LIN {X 0,Y 369.216,Z 142.49,A -85,B 0,C 180,E1 -12872.663,E2 -12872.663} C_VEL
LIN {X 0,Y 369.197,Z 142.498,A -85,B 0,C 180,E1 -12876.558,E2 -12876.558} C_VEL
LIN {X 0,Y 369.156,Z 142.497,A -85,B 0,C 180,E1 -12877.428,E2 -12877.428} C_VEL
LIN {X 0,Y 368.474,Z 142.588,A -85,B 0,C 180,E1 -12878.338,E2 -12878.338} C_VEL
LIN {X 0,Y 365.538,Z 142.949,A -85,B 0,C 180,E1 -12879.815,E2 -12879.815} C_VEL
LIN {X 0,Y 363.064,Z 143.259,A -85,B 0,C 180,E1 -12881.01,E2 -12881.01} C_VEL
LIN {X 0,Y 362.026,Z 143.387,A -85,B 0,C 180,E1 -12881.936,E2 -12881.936} C_VEL
LIN {X 0,Y 361.954,Z 143.398,A -85,B 0,C 180,E1 -12882.25,E2 -12882.25} C_VEL
LIN {X 0,Y 361.96,Z 143.399,A -85,B 0,C 180,E1 -12884.62,E2 -12884.62} C_VEL
LIN {X 0,Y 361.957,Z 143.398,A -85,B 0,C 180,E1 -12888.099,E2 -12888.099} C_VEL
LIN {X 0,Y 361.859,Z 143.407,A -85,B 0,C 180,E1 -12891.654,E2 -12891.654} C_VEL
LIN {X 0,Y 361.924,Z 143.399,A -85,B 0,C 180,E1 -12895.29,E2 -12895.29} C_VEL
LIN {X 0,Y 361.919,Z 143.401,A -85,B 0,C 180,E1 -12897.778,E2 -12897.778} C_VEL
LIN {X 0,Y 361.856,Z 143.409,A -85,B 0,C 180,E1 -12901.627,E2 -12901.627} C_VEL
LIN {X 0,Y 361.871,Z 143.406,A -85,B 0,C 180,E1 -12905.345,E2 -12905.345} C_VEL
LIN {X 0,Y 361.869,Z 143.406,A -85,B 0,C 180,E1 -12909.027,E2 -12909.027} C_VEL
LIN {X 0,Y 361.88,Z 143.406,A -85,B 0,C 180,E1 -12912.44,E2 -12912.44} C_VEL
LIN {X 0,Y 361.862,Z 143.411,A -85,B 0,C 180,E1 -12915.639,E2 -12915.639} C_VEL
LIN {X 0,Y 361.869,Z 143.407,A -85,B 0,C 180,E1 -12919.238,E2 -12919.238} C_VEL
LIN {X 0,Y 361.866,Z 143.407,A -85,B 0,C 180,E1 -12922.982,E2 -12922.982} C_VEL
LIN {X 0,Y 361.857,Z 143.407,A -85,B 0,C 180,E1 -12926.63,E2 -12926.63} C_VEL
LIN {X 0,Y 361.871,Z 143.41,A -85,B 0,C 180,E1 -12929.672,E2 -12929.672} C_VEL
LIN {X 0,Y 361.951,Z 143.401,A -85,B 0,C 180,E1 -12933.475,E2 -12933.475} C_VEL
LIN {X 0,Y 361.887,Z 143.407,A -85,B 0,C 180,E1 -12937.145,E2 -12937.145} C_VEL
LIN {X 0,Y 361.918,Z 143.401,A -85,B 0,C 180,E1 -12940.724,E2 -12940.724} C_VEL
LIN {X 0,Y 361.943,Z 143.396,A -85,B 0,C 180,E1 -12944.226,E2 -12944.226} C_VEL
LIN {X 0,Y 361.996,Z 143.391,A -85,B 0,C 180,E1 -12946.528,E2 -12946.528} C_VEL
LIN {X 0,Y 362.029,Z 143.386,A -85,B 0,C 180,E1 -12949.938,E2 -12949.938} C_VEL
LIN {X 0,Y 362.158,Z 143.373,A -85,B 0,C 180,E1 -12953.314,E2 -12953.314} C_VEL
LIN {X 0,Y 362.281,Z 143.354,A -85,B 0,C 180,E1 -12957.777,E2 -12957.777} C_VEL
LIN {X 0,Y 362.426,Z 143.336,A -85,B 0,C 180,E1 -12960,E2 -12960} C_VEL
LIN {X 0,Y 362.281,Z 143.355,A -85,B 0,C 180,E1 -12962.224,E2 -12962.224} C_VEL
LIN {X 0,Y 362.171,Z 143.374,A -85,B 0,C 180,E1 -12966.687,E2 -12966.687} C_VEL
LIN {X 0,Y 362.072,Z 143.384,A -85,B 0,C 180,E1 -12968.934,E2 -12968.934} C_VEL
LIN {X 0,Y 361.959,Z 143.398,A -85,B 0,C 180,E1 -12972.333,E2 -12972.333} C_VEL
LIN {X 0,Y 361.961,Z 143.4,A -85,B 0,C 180,E1 -12974.621,E2 -12974.621} C_VEL
LIN {X 0,Y 361.958,Z 143.397,A -85,B 0,C 180,E1 -12978.1,E2 -12978.1} C_VEL
LIN {X 0,Y 361.86,Z 143.407,A -85,B 0,C 180,E1 -12981.655,E2 -12981.655} C_VEL
LIN {X 0,Y 361.925,Z 143.398,A -85,B 0,C 180,E1 -12985.291,E2 -12985.291} C_VEL
LIN {X 0,Y 361.917,Z 143.401,A -85,B 0,C 180,E1 -12987.779,E2 -12987.779} C_VEL
LIN {X 0,Y 361.846,Z 143.408,A -85,B 0,C 180,E1 -12991.286,E2 -12991.286} C_VEL
LIN {X 0,Y 361.854,Z 143.412,A -85,B 0,C 180,E1 -12994.281,E2 -12994.281} C_VEL
LIN {X 0,Y 361.865,Z 143.406,A -85,B 0,C 180,E1 -12997.224,E2 -12997.224} C_VEL
LIN {X 0,Y 361.872,Z 143.405,A -85,B 0,C 180,E1 -13000.763,E2 -13000.763} C_VEL
LIN {X 0,Y 361.822,Z 143.413,A -85,B 0,C 180,E1 -13004.368,E2 -13004.368} C_VEL
LIN {X 0,Y 361.836,Z 143.413,A -85,B 0,C 180,E1 -13007.569,E2 -13007.569} C_VEL
LIN {X 0,Y 361.869,Z 143.406,A -85,B 0,C 180,E1 -13010.974,E2 -13010.974} C_VEL
LIN {X 0,Y 361.875,Z 143.405,A -85,B 0,C 180,E1 -13014.656,E2 -13014.656} C_VEL
LIN {X 0,Y 361.838,Z 143.412,A -85,B 0,C 180,E1 -13018.371,E2 -13018.371} C_VEL
LIN {X 0,Y 361.909,Z 143.415,A -85,B 0,C 180,E1 -13019.6,E2 -13019.6} C_VEL
LIN {X 0,Y 364.625,Z 156.408,A -85,B 0,C 180,E1 -13022.671,E2 -13022.671} C_VEL
LIN {X 0,Y 365.599,Z 162.364,A -85,B 0,C 180,E1 -13024.029,E2 -13024.029} C_VEL
LIN {X 0,Y 364.449,Z 176.387,A -85,B 0,C 180,E1 -13027.015,E2 -13027.015} C_VEL
LIN {X 0,Y 363.824,Z 184.769,A -85,B 0,C 180,E1 -13028.787,E2 -13028.787} C_VEL
LIN {X 0,Y 368.173,Z 221.285,A -85,B 0,C 180,E1 -13029.864,E2 -13029.864} C_VEL
LIN {X 0,Y 366.668,Z 294.38,A -85,B 0,C 180,E1 -13031.564,E2 -13031.564} C_VEL
LIN {X 0,Y 365.977,Z 308.139,A -85,B 0,C 180,E1 -13032.107,E2 -13032.107} C_VEL
LIN {X 0,Y 365.231,Z 320.13,A -85,B 0,C 180,E1 -13032.792,E2 -13032.792} C_VEL
LIN {X 0,Y 364.244,Z 332.659,A -85,B 0,C 180,E1 -13033.754,E2 -13033.754} C_VEL
LIN {X 0,Y 363.427,Z 343.96,A -85,B 0,C 180,E1 -13034.867,E2 -13034.867} C_VEL
LIN {X 0,Y 362.616,Z 353.865,A -85,B 0,C 180,E1 -13036.083,E2 -13036.083} C_VEL
LIN {X 0,Y 361.884,Z 364.213,A -85,B 0,C 180,E1 -13037.665,E2 -13037.665} C_VEL
LIN {X 0,Y 361.231,Z 371.672,A -85,B 0,C 180,E1 -13039.066,E2 -13039.066} C_VEL
LIN {X 0,Y 360.793,Z 378.999,A -85,B 0,C 180,E1 -13040.753,E2 -13040.753} C_VEL
LIN {X 0,Y 360.628,Z 383.937,A -85,B 0,C 180,E1 -13042.16,E2 -13042.16} C_VEL
LIN {X 0,Y 360.458,Z 388.862,A -85,B 0,C 180,E1 -13043.92,E2 -13043.92} C_VEL
LIN {X 0,Y 360.482,Z 392.245,A -85,B 0,C 180,E1 -13045.528,E2 -13045.528} C_VEL
LIN {X 0,Y 360.417,Z 393.997,A -85,B 0,C 180,E1 -13046.647,E2 -13046.647} C_VEL
LIN {X 0,Y 360.545,Z 395.32,A -85,B 0,C 180,E1 -13047.766,E2 -13047.766} C_VEL
LIN {X 0,Y 360.539,Z 396.212,A -85,B 0,C 180,E1 -13048.883,E2 -13048.883} C_VEL
LIN {X 0,Y 360.527,Z 396.662,A -85,B 0,C 180,E1 -13050,E2 -13050} C_VEL
LIN {X 0,Y 360.516,Z 396.658,A -85,B 0,C 180,E1 -13051.117,E2 -13051.117} C_VEL
LIN {X 0,Y 360.429,Z 396.239,A -85,B 0,C 180,E1 -13052.235,E2 -13052.235} C_VEL
LIN {X 0,Y 360.366,Z 395.415,A -85,B 0,C 180,E1 -13053.355,E2 -13053.355} C_VEL
LIN {X 0,Y 360.383,Z 394.141,A -85,B 0,C 180,E1 -13054.474,E2 -13054.474} C_VEL
LIN {X 0,Y 360.318,Z 391.949,A -85,B 0,C 180,E1 -13055.868,E2 -13055.868} C_VEL
LIN {X 0,Y 360.598,Z 387.648,A -85,B 0,C 180,E1 -13057.842,E2 -13057.842} C_VEL
LIN {X 0,Y 360.929,Z 382.737,A -85,B 0,C 180,E1 -13059.527,E2 -13059.527} C_VEL
LIN {X 0,Y 361.665,Z 375.38,A -85,B 0,C 180,E1 -13061.489,E2 -13061.489} C_VEL
LIN {X 0,Y 362.609,Z 367.453,A -85,B 0,C 180,E1 -13063.164,E2 -13063.164} C_VEL
LIN {X 0,Y 363.547,Z 358.621,A -85,B 0,C 180,E1 -13064.675,E2 -13064.675} C_VEL
LIN {X 0,Y 364.773,Z 348.543,A -85,B 0,C 180,E1 -13066.079,E2 -13066.079} C_VEL
LIN {X 0,Y 366.12,Z 337.576,A -85,B 0,C 180,E1 -13067.31,E2 -13067.31} C_VEL
LIN {X 0,Y 367.554,Z 325.219,A -85,B 0,C 180,E1 -13068.391,E2 -13068.391} C_VEL
LIN {X 0,Y 368.706,Z 312.247,A -85,B 0,C 180,E1 -13069.269,E2 -13069.269} C_VEL
LIN {X 0,Y 369.888,Z 298.194,A -85,B 0,C 180,E1 -13069.927,E2 -13069.927} C_VEL
LIN {X 0,Y 370.467,Z 285.445,A -85,B 0,C 180,E1 -13070.329,E2 -13070.329} C_VEL
LIN {X 0,Y 372.333,Z 220.719,A -85,B 0,C 180,E1 -13071.896,E2 -13071.896} C_VEL
LIN {X 0,Y 370.378,Z 204.902,A -85,B 0,C 180,E1 -13072.497,E2 -13072.497} C_VEL
LIN {X 0,Y 367.323,Z 188.483,A -85,B 0,C 180,E1 -13073.223,E2 -13073.223} C_VEL
LIN {X 0,Y 365.724,Z 180.687,A -85,B 0,C 180,E1 -13073.613,E2 -13073.613} C_VEL
LIN {X 0,Y 367.221,Z 166.298,A -85,B 0,C 180,E1 -13076.728,E2 -13076.728} C_VEL
LIN {X 0,Y 365.197,Z 156.175,A -85,B 0,C 180,E1 -13079.289,E2 -13079.289} C_VEL
LIN {X 0,Y 362.447,Z 145.496,A -85,B 0,C 180,E1 -13082.224,E2 -13082.224} C_VEL
LIN {X 0,Y 361.868,Z 143.412,A -85,B 0,C 180,E1 -13082.86,E2 -13082.86} C_VEL
LIN {X 0,Y 361.872,Z 143.409,A -85,B 0,C 180,E1 -13085.637,E2 -13085.637} C_VEL
LIN {X 0,Y 361.874,Z 143.41,A -85,B 0,C 180,E1 -13089.027,E2 -13089.027} C_VEL
LIN {X 0,Y 361.84,Z 143.413,A -85,B 0,C 180,E1 -13092.829,E2 -13092.829} C_VEL
LIN {X 0,Y 361.821,Z 143.412,A -85,B 0,C 180,E1 -13095.947,E2 -13095.947} C_VEL
LIN {X 0,Y 361.839,Z 143.408,A -85,B 0,C 180,E1 -13099.245,E2 -13099.245} C_VEL
LIN {X 0,Y 361.866,Z 143.404,A -85,B 0,C 180,E1 -13102.777,E2 -13102.777} C_VEL
LIN {X 0,Y 361.857,Z 143.404,A -85,B 0,C 180,E1 -13105.719,E2 -13105.719} C_VEL
LIN {X 0,Y 361.876,Z 143.408,A -85,B 0,C 180,E1 -13109.672,E2 -13109.672} C_VEL
LIN {X 0,Y 361.957,Z 143.396,A -85,B 0,C 180,E1 -13113.475,E2 -13113.475} C_VEL
LIN {X 0,Y 361.894,Z 143.402,A -85,B 0,C 180,E1 -13117.145,E2 -13117.145} C_VEL
LIN {X 0,Y 361.907,Z 143.404,A -85,B 0,C 180,E1 -13120.723,E2 -13120.723} C_VEL
LIN {X 0,Y 361.946,Z 143.396,A -85,B 0,C 180,E1 -13124.226,E2 -13124.226} C_VEL
LIN {X 0,Y 362.002,Z 143.391,A -85,B 0,C 180,E1 -13126.528,E2 -13126.528} C_VEL
LIN {X 0,Y 362.003,Z 143.393,A -85,B 0,C 180,E1 -13129.937,E2 -13129.937} C_VEL
LIN {X 0,Y 362.138,Z 143.38,A -85,B 0,C 180,E1 -13133.313,E2 -13133.313} C_VEL
LIN {X 0,Y 362.28,Z 143.363,A -85,B 0,C 180,E1 -13137.776,E2 -13137.776} C_VEL
LIN {X 0,Y 362.271,Z 143.399,A -85,B 0,C 180,E1 -13139.374,E2 -13139.374} C_VEL
LIN {X 0,Y 363.828,Z 149.687,A -85,B 0,C 180,E1 -13141.279,E2 -13141.279} C_VEL
LIN {X 0,Y 369.872,Z 162.966,A -85,B 0,C 180,E1 -13142.249,E2 -13142.249} C_VEL
LIN {X 0,Y 373.599,Z 171.886,A -85,B 0,C 180,E1 -13142.827,E2 -13142.827} C_VEL
LIN {X 0,Y 373.603,Z 177.913,A -85,B 0,C 180,E1 -13142.993,E2 -13142.993} C_VEL
LIN {X 0,Y 370.924,Z 256.422,A -85,B 0,C 180,E1 -13144.925,E2 -13144.925} C_VEL
LIN {X 0,Y 370.325,Z 269.377,A -85,B 0,C 180,E1 -13145.445,E2 -13145.445} C_VEL
LIN {X 0,Y 369.501,Z 282.588,A -85,B 0,C 180,E1 -13146.21,E2 -13146.21} C_VEL
LIN {X 0,Y 368.37,Z 295.305,A -85,B 0,C 180,E1 -13147.21,E2 -13147.21} C_VEL
LIN {X 0,Y 367.186,Z 306.94,A -85,B 0,C 180,E1 -13148.392,E2 -13148.392} C_VEL
LIN {X 0,Y 366.046,Z 316.914,A -85,B 0,C 180,E1 -13149.671,E2 -13149.671} C_VEL
LIN {X 0,Y 364.896,Z 326.008,A -85,B 0,C 180,E1 -13151.104,E2 -13151.104} C_VEL
LIN {X 0,Y 363.882,Z 333.5,A -85,B 0,C 180,E1 -13152.549,E2 -13152.549} C_VEL
LIN {X 0,Y 363.102,Z 339.353,A -85,B 0,C 180,E1 -13153.919,E2 -13153.919} C_VEL
LIN {X 0,Y 362.234,Z 345.726,A -85,B 0,C 180,E1 -13155.761,E2 -13155.761} C_VEL
LIN {X 0,Y 361.527,Z 350.802,A -85,B 0,C 180,E1 -13157.72,E2 -13157.72} C_VEL
LIN {X 0,Y 361.079,Z 353.856,A -85,B 0,C 180,E1 -13159.322,E2 -13159.322} C_VEL
LIN {X 0,Y 360.773,Z 355.83,A -85,B 0,C 180,E1 -13160.761,E2 -13160.761} C_VEL
LIN {X 0,Y 360.607,Z 356.736,A -85,B 0,C 180,E1 -13161.734,E2 -13161.734} C_VEL
LIN {X 0,Y 360.406,Z 357.591,A -85,B 0,C 180,E1 -13163.578,E2 -13163.578} C_VEL
LIN {X 0,Y 360.338,Z 357.323,A -85,B 0,C 180,E1 -13165.409,E2 -13165.409} C_VEL
LIN {X 0,Y 360.335,Z 356.51,A -85,B 0,C 180,E1 -13166.653,E2 -13166.653} C_VEL
LIN {X 0,Y 360.495,Z 354.072,A -85,B 0,C 180,E1 -13168.682,E2 -13168.682} C_VEL
LIN {X 0,Y 360.795,Z 350.782,A -85,B 0,C 180,E1 -13170.428,E2 -13170.428} C_VEL
LIN {X 0,Y 361.1,Z 345.75,A -85,B 0,C 180,E1 -13172.359,E2 -13172.359} C_VEL
LIN {X 0,Y 361.657,Z 339.068,A -85,B 0,C 180,E1 -13174.301,E2 -13174.301} C_VEL
LIN {X 0,Y 362.212,Z 331.861,A -85,B 0,C 180,E1 -13175.94,E2 -13175.94} C_VEL
LIN {X 0,Y 362.867,Z 323.153,A -85,B 0,C 180,E1 -13177.54,E2 -13177.54} C_VEL
LIN {X 0,Y 363.717,Z 313.001,A -85,B 0,C 180,E1 -13179.043,E2 -13179.043} C_VEL
LIN {X 0,Y 364.558,Z 301.376,A -85,B 0,C 180,E1 -13180.408,E2 -13180.408} C_VEL
LIN {X 0,Y 365.294,Z 291.019,A -85,B 0,C 180,E1 -13181.38,E2 -13181.38} C_VEL
LIN {X 0,Y 365.95,Z 279.585,A -85,B 0,C 180,E1 -13182.234,E2 -13182.234} C_VEL
LIN {X 0,Y 366.468,Z 266.205,A -85,B 0,C 180,E1 -13182.978,E2 -13182.978} C_VEL
LIN {X 0,Y 366.947,Z 253.458,A -85,B 0,C 180,E1 -13183.461,E2 -13183.461} C_VEL
LIN {X 0,Y 368.802,Z 168.805,A -85,B 0,C 180,E1 -13185.403,E2 -13185.403} C_VEL
LIN {X 0,Y 366.602,Z 159.202,A -85,B 0,C 180,E1 -13185.738,E2 -13185.738} C_VEL
LIN {X 0,Y 362.416,Z 146.013,A -85,B 0,C 180,E1 -13186.279,E2 -13186.279} C_VEL
LIN {X 0,Y 361.912,Z 143.405,A -85,B 0,C 180,E1 -13186.992,E2 -13186.992} C_VEL
LIN {X 0,Y 361.867,Z 143.406,A -85,B 0,C 180,E1 -13190.973,E2 -13190.973} C_VEL
LIN {X 0,Y 361.873,Z 143.405,A -85,B 0,C 180,E1 -13194.655,E2 -13194.655} C_VEL
LIN {X 0,Y 361.836,Z 143.41,A -85,B 0,C 180,E1 -13198.37,E2 -13198.37} C_VEL
LIN {X 0,Y 361.899,Z 143.403,A -85,B 0,C 180,E1 -13200.955,E2 -13200.955} C_VEL
LIN {X 0,Y 361.954,Z 143.4,A -85,B 0,C 180,E1 -13203.475,E2 -13203.475} C_VEL
LIN {X 0,Y 361.89,Z 143.408,A -85,B 0,C 180,E1 -13207.144,E2 -13207.144} C_VEL
LIN {X 0,Y 361.885,Z 143.405,A -85,B 0,C 180,E1 -13210.722,E2 -13210.722} C_VEL
LIN {X 0,Y 361.942,Z 143.396,A -85,B 0,C 180,E1 -13214.226,E2 -13214.226} C_VEL
LIN {X 0,Y 361.998,Z 143.391,A -85,B 0,C 180,E1 -13216.527,E2 -13216.527} C_VEL
LIN {X 0,Y 362.03,Z 143.385,A -85,B 0,C 180,E1 -13219.938,E2 -13219.938} C_VEL
LIN {X 0,Y 362.159,Z 143.372,A -85,B 0,C 180,E1 -13223.313,E2 -13223.313} C_VEL
LIN {X 0,Y 362.281,Z 143.354,A -85,B 0,C 180,E1 -13227.776,E2 -13227.776} C_VEL
LIN {X 0,Y 362.427,Z 143.336,A -85,B 0,C 180,E1 -13230,E2 -13230} C_VEL
LIN {X 0,Y 362.281,Z 143.356,A -85,B 0,C 180,E1 -13232.223,E2 -13232.223} C_VEL
LIN {X 0,Y 362.159,Z 143.376,A -85,B 0,C 180,E1 -13236.686,E2 -13236.686} C_VEL
LIN {X 0,Y 362.029,Z 143.387,A -85,B 0,C 180,E1 -13240.062,E2 -13240.062} C_VEL
LIN {X 0,Y 361.954,Z 143.398,A -85,B 0,C 180,E1 -13242.25,E2 -13242.25} C_VEL
LIN {X 0,Y 361.309,Z 143.484,A -85,B 0,C 180,E1 -13243.179,E2 -13243.179} C_VEL
LIN {X 0,Y 358.42,Z 143.841,A -85,B 0,C 180,E1 -13244.687,E2 -13244.687} C_VEL
LIN {X 0,Y 355.975,Z 144.141,A -85,B 0,C 180,E1 -13245.908,E2 -13245.908} C_VEL
LIN {X 0,Y 354.955,Z 144.269,A -85,B 0,C 180,E1 -13246.854,E2 -13246.854} C_VEL
LIN {X 0,Y 354.889,Z 144.275,A -85,B 0,C 180,E1 -13247.174,E2 -13247.174} C_VEL
LIN {X 0,Y 354.863,Z 144.279,A -85,B 0,C 180,E1 -13249.674,E2 -13249.674} C_VEL
LIN {X 0,Y 354.824,Z 144.283,A -85,B 0,C 180,E1 -13253.337,E2 -13253.337} C_VEL
LIN {X 0,Y 354.886,Z 144.276,A -85,B 0,C 180,E1 -13256.982,E2 -13256.982} C_VEL
LIN {X 0,Y 354.851,Z 144.281,A -85,B 0,C 180,E1 -13259.678,E2 -13259.678} C_VEL
LIN {X 0,Y 354.827,Z 144.285,A -85,B 0,C 180,E1 -13263.682,E2 -13263.682} C_VEL
LIN {X 0,Y 354.796,Z 144.289,A -85,B 0,C 180,E1 -13266.459,E2 -13266.459} C_VEL
LIN {X 0,Y 354.82,Z 144.285,A -85,B 0,C 180,E1 -13269.423,E2 -13269.423} C_VEL
LIN {X 0,Y 354.832,Z 144.282,A -85,B 0,C 180,E1 -13272.875,E2 -13272.875} C_VEL
LIN {X 0,Y 354.801,Z 144.289,A -85,B 0,C 180,E1 -13276.109,E2 -13276.109} C_VEL
LIN {X 0,Y 354.821,Z 144.285,A -85,B 0,C 180,E1 -13279.184,E2 -13279.184} C_VEL
LIN {X 0,Y 354.805,Z 144.286,A -85,B 0,C 180,E1 -13282.402,E2 -13282.402} C_VEL
LIN {X 0,Y 354.809,Z 144.286,A -85,B 0,C 180,E1 -13284.941,E2 -13284.941} C_VEL
LIN {X 0,Y 354.791,Z 144.287,A -85,B 0,C 180,E1 -13288.405,E2 -13288.405} C_VEL
LIN {X 0,Y 354.847,Z 144.285,A -85,B 0,C 180,E1 -13291.619,E2 -13291.619} C_VEL
LIN {X 0,Y 354.896,Z 144.275,A -85,B 0,C 180,E1 -13294.173,E2 -13294.173} C_VEL
LIN {X 0,Y 354.832,Z 144.284,A -85,B 0,C 180,E1 -13297.894,E2 -13297.894} C_VEL
LIN {X 0,Y 354.92,Z 144.272,A -85,B 0,C 180,E1 -13301.892,E2 -13301.892} C_VEL
LIN {X 0,Y 354.94,Z 144.269,A -85,B 0,C 180,E1 -13305.981,E2 -13305.981} C_VEL
LIN {X 0,Y 354.976,Z 144.265,A -85,B 0,C 180,E1 -13309.736,E2 -13309.736} C_VEL
LIN {X 0,Y 355.123,Z 144.25,A -85,B 0,C 180,E1 -13313.181,E2 -13313.181} C_VEL
LIN {X 0,Y 355.244,Z 144.231,A -85,B 0,C 180,E1 -13317.733,E2 -13317.733} C_VEL
LIN {X 0,Y 355.396,Z 144.212,A -85,B 0,C 180,E1 -13320,E2 -13320} C_VEL
LIN {X 0,Y 355.244,Z 144.232,A -85,B 0,C 180,E1 -13322.268,E2 -13322.268} C_VEL
LIN {X 0,Y 355.137,Z 144.249,A -85,B 0,C 180,E1 -13326.82,E2 -13326.82} C_VEL
LIN {X 0,Y 355.014,Z 144.262,A -85,B 0,C 180,E1 -13329.113,E2 -13329.113} C_VEL
LIN {X 0,Y 354.92,Z 144.277,A -85,B 0,C 180,E1 -13332.581,E2 -13332.581} C_VEL
LIN {X 0,Y 354.889,Z 144.277,A -85,B 0,C 180,E1 -13336.096,E2 -13336.096} C_VEL
LIN {X 0,Y 354.905,Z 144.279,A -85,B 0,C 180,E1 -13338.472,E2 -13338.472} C_VEL
LIN {X 0,Y 354.815,Z 144.288,A -85,B 0,C 180,E1 -13342.108,E2 -13342.108} C_VEL
LIN {X 0,Y 354.897,Z 144.276,A -85,B 0,C 180,E1 -13345.828,E2 -13345.828} C_VEL
LIN {X 0,Y 354.853,Z 144.281,A -85,B 0,C 180,E1 -13349.679,E2 -13349.679} C_VEL
LIN {X 0,Y 354.805,Z 144.287,A -85,B 0,C 180,E1 -13353.703,E2 -13353.703} C_VEL
LIN {X 0,Y 354.799,Z 144.289,A -85,B 0,C 180,E1 -13356.46,E2 -13356.46} C_VEL
LIN {X 0,Y 354.824,Z 144.284,A -85,B 0,C 180,E1 -13359.424,E2 -13359.424} C_VEL
LIN {X 0,Y 354.804,Z 144.286,A -85,B 0,C 180,E1 -13362.871,E2 -13362.871} C_VEL
LIN {X 0,Y 354.768,Z 144.294,A -85,B 0,C 180,E1 -13366.104,E2 -13366.104} C_VEL
LIN {X 0,Y 354.788,Z 144.288,A -85,B 0,C 180,E1 -13369.18,E2 -13369.18} C_VEL
LIN {X 0,Y 354.808,Z 144.286,A -85,B 0,C 180,E1 -13372.403,E2 -13372.403} C_VEL
LIN {X 0,Y 354.812,Z 144.285,A -85,B 0,C 180,E1 -13374.941,E2 -13374.941} C_VEL
LIN {X 0,Y 354.826,Z 144.287,A -85,B 0,C 180,E1 -13379.005,E2 -13379.005} C_VEL
LIN {X 0,Y 354.893,Z 144.446,A -85,B 0,C 180,E1 -13379.383,E2 -13379.383} C_VEL
LIN {X 0,Y 357.935,Z 159.065,A -85,B 0,C 180,E1 -13382.895,E2 -13382.895} C_VEL
LIN {X 0,Y 358.604,Z 164.655,A -85,B 0,C 180,E1 -13384.179,E2 -13384.179} C_VEL
LIN {X 0,Y 356.86,Z 184.383,A -85,B 0,C 180,E1 -13388.445,E2 -13388.445} C_VEL
LIN {X 0,Y 361.314,Z 221.994,A -85,B 0,C 180,E1 -13389.591,E2 -13389.591} C_VEL
LIN {X 0,Y 359.764,Z 294.104,A -85,B 0,C 180,E1 -13391.308,E2 -13391.308} C_VEL
LIN {X 0,Y 359.082,Z 307.818,A -85,B 0,C 180,E1 -13391.862,E2 -13391.862} C_VEL
LIN {X 0,Y 358.264,Z 320.276,A -85,B 0,C 180,E1 -13392.594,E2 -13392.594} C_VEL
LIN {X 0,Y 357.251,Z 332.695,A -85,B 0,C 180,E1 -13393.574,E2 -13393.574} C_VEL
LIN {X 0,Y 356.409,Z 343.919,A -85,B 0,C 180,E1 -13394.708,E2 -13394.708} C_VEL
LIN {X 0,Y 355.516,Z 354.668,A -85,B 0,C 180,E1 -13396.08,E2 -13396.08} C_VEL
LIN {X 0,Y 354.749,Z 364.889,A -85,B 0,C 180,E1 -13397.704,E2 -13397.704} C_VEL
LIN {X 0,Y 354.024,Z 373.445,A -85,B 0,C 180,E1 -13399.419,E2 -13399.419} C_VEL
LIN {X 0,Y 353.682,Z 380.33,A -85,B 0,C 180,E1 -13401.142,E2 -13401.142} C_VEL
LIN {X 0,Y 353.397,Z 386.57,A -85,B 0,C 180,E1 -13403.147,E2 -13403.147} C_VEL
LIN {X 0,Y 353.384,Z 390.579,A -85,B 0,C 180,E1 -13404.866,E2 -13404.866} C_VEL
LIN {X 0,Y 353.335,Z 393.476,A -85,B 0,C 180,E1 -13406.579,E2 -13406.579} C_VEL
LIN {X 0,Y 353.447,Z 394.825,A -85,B 0,C 180,E1 -13407.721,E2 -13407.721} C_VEL
LIN {X 0,Y 353.475,Z 395.745,A -85,B 0,C 180,E1 -13408.861,E2 -13408.861} C_VEL
LIN {X 0,Y 353.462,Z 396.241,A -85,B 0,C 180,E1 -13410,E2 -13410} C_VEL
LIN {X 0,Y 353.432,Z 396.269,A -85,B 0,C 180,E1 -13411.14,E2 -13411.14} C_VEL
LIN {X 0,Y 353.33,Z 395.877,A -85,B 0,C 180,E1 -13412.28,E2 -13412.28} C_VEL
LIN {X 0,Y 353.282,Z 395.078,A -85,B 0,C 180,E1 -13413.422,E2 -13413.422} C_VEL
LIN {X 0,Y 353.289,Z 393.855,A -85,B 0,C 180,E1 -13414.564,E2 -13414.564} C_VEL
LIN {X 0,Y 353.235,Z 391.94,A -85,B 0,C 180,E1 -13415.838,E2 -13415.838} C_VEL
LIN {X 0,Y 353.53,Z 387.454,A -85,B 0,C 180,E1 -13417.999,E2 -13417.999} C_VEL
LIN {X 0,Y 353.908,Z 382.601,A -85,B 0,C 180,E1 -13419.718,E2 -13419.718} C_VEL
LIN {X 0,Y 354.688,Z 375.317,A -85,B 0,C 180,E1 -13421.719,E2 -13421.719} C_VEL
LIN {X 0,Y 355.689,Z 367.504,A -85,B 0,C 180,E1 -13423.425,E2 -13423.425} C_VEL
LIN {X 0,Y 356.694,Z 358.553,A -85,B 0,C 180,E1 -13425.009,E2 -13425.009} C_VEL
LIN {X 0,Y 358.122,Z 347.778,A -85,B 0,C 180,E1 -13426.533,E2 -13426.533} C_VEL
LIN {X 0,Y 359.558,Z 336.707,A -85,B 0,C 180,E1 -13427.783,E2 -13427.783} C_VEL
LIN {X 0,Y 361.039,Z 324.241,A -85,B 0,C 180,E1 -13428.883,E2 -13428.883} C_VEL
LIN {X 0,Y 362.179,Z 312.245,A -85,B 0,C 180,E1 -13429.704,E2 -13429.704} C_VEL
LIN {X 0,Y 363.414,Z 298.533,A -85,B 0,C 180,E1 -13430.371,E2 -13430.371} C_VEL
LIN {X 0,Y 364.071,Z 285.149,A -85,B 0,C 180,E1 -13430.813,E2 -13430.813} C_VEL
LIN {X 0,Y 366.037,Z 221.315,A -85,B 0,C 180,E1 -13432.406,E2 -13432.406} C_VEL
LIN {X 0,Y 364.169,Z 206.128,A -85,B 0,C 180,E1 -13433,E2 -13433} C_VEL
LIN {X 0,Y 360.866,Z 188.359,A -85,B 0,C 180,E1 -13433.827,E2 -13433.827} C_VEL
LIN {X 0,Y 359.191,Z 180.15,A -85,B 0,C 180,E1 -13434.261,E2 -13434.261} C_VEL
LIN {X 0,Y 360.437,Z 167.993,A -85,B 0,C 180,E1 -13436.959,E2 -13436.959} C_VEL
LIN {X 0,Y 358.62,Z 158.852,A -85,B 0,C 180,E1 -13439.337,E2 -13439.337} C_VEL
LIN {X 0,Y 356.06,Z 148.667,A -85,B 0,C 180,E1 -13442.204,E2 -13442.204} C_VEL
LIN {X 0,Y 354.815,Z 144.29,A -85,B 0,C 180,E1 -13443.558,E2 -13443.558} C_VEL
LIN {X 0,Y 354.802,Z 144.291,A -85,B 0,C 180,E1 -13446.459,E2 -13446.459} C_VEL
LIN {X 0,Y 354.828,Z 144.289,A -85,B 0,C 180,E1 -13449.424,E2 -13449.424} C_VEL
LIN {X 0,Y 354.792,Z 144.291,A -85,B 0,C 180,E1 -13452.867,E2 -13452.867} C_VEL
LIN {X 0,Y 354.77,Z 144.29,A -85,B 0,C 180,E1 -13456.104,E2 -13456.104} C_VEL
LIN {X 0,Y 354.791,Z 144.285,A -85,B 0,C 180,E1 -13459.179,E2 -13459.179} C_VEL
LIN {X 0,Y 354.81,Z 144.284,A -85,B 0,C 180,E1 -13462.403,E2 -13462.403} C_VEL
LIN {X 0,Y 354.815,Z 144.284,A -85,B 0,C 180,E1 -13464.941,E2 -13464.941} C_VEL
LIN {X 0,Y 354.796,Z 144.283,A -85,B 0,C 180,E1 -13468.405,E2 -13468.405} C_VEL
LIN {X 0,Y 354.85,Z 144.279,A -85,B 0,C 180,E1 -13471.618,E2 -13471.618} C_VEL
LIN {X 0,Y 354.903,Z 144.27,A -85,B 0,C 180,E1 -13474.172,E2 -13474.172} C_VEL
LIN {X 0,Y 354.838,Z 144.284,A -85,B 0,C 180,E1 -13477.894,E2 -13477.894} C_VEL
LIN {X 0,Y 354.893,Z 144.272,A -85,B 0,C 180,E1 -13481.908,E2 -13481.908} C_VEL
LIN {X 0,Y 354.946,Z 144.271,A -85,B 0,C 180,E1 -13485.981,E2 -13485.981} C_VEL
LIN {X 0,Y 354.959,Z 144.271,A -85,B 0,C 180,E1 -13489.735,E2 -13489.735} C_VEL
LIN {X 0,Y 355.103,Z 144.257,A -85,B 0,C 180,E1 -13493.18,E2 -13493.18} C_VEL
LIN {X 0,Y 355.243,Z 144.239,A -85,B 0,C 180,E1 -13497.732,E2 -13497.732} C_VEL
LIN {X 0,Y 355.213,Z 144.411,A -85,B 0,C 180,E1 -13498.724,E2 -13498.724} C_VEL
LIN {X 0,Y 356.811,Z 150.318,A -85,B 0,C 180,E1 -13500.585,E2 -13500.585} C_VEL
LIN {X 0,Y 362.801,Z 162.829,A -85,B 0,C 180,E1 -13501.572,E2 -13501.572} C_VEL
LIN {X 0,Y 367.561,Z 173.93,A -85,B 0,C 180,E1 -13502.353,E2 -13502.353} C_VEL
LIN {X 0,Y 364.521,Z 257.464,A -85,B 0,C 180,E1 -13504.457,E2 -13504.457} C_VEL
LIN {X 0,Y 363.854,Z 270.838,A -85,B 0,C 180,E1 -13505.021,E2 -13505.021} C_VEL
LIN {X 0,Y 363.039,Z 283.148,A -85,B 0,C 180,E1 -13505.763,E2 -13505.763} C_VEL
LIN {X 0,Y 361.943,Z 294.792,A -85,B 0,C 180,E1 -13506.69,E2 -13506.69} C_VEL
LIN {X 0,Y 360.745,Z 306.127,A -85,B 0,C 180,E1 -13507.838,E2 -13507.838} C_VEL
LIN {X 0,Y 359.513,Z 316.389,A -85,B 0,C 180,E1 -13509.139,E2 -13509.139} C_VEL
LIN {X 0,Y 358.295,Z 325.525,A -85,B 0,C 180,E1 -13510.575,E2 -13510.575} C_VEL
LIN {X 0,Y 357.088,Z 333.981,A -85,B 0,C 180,E1 -13512.214,E2 -13512.214} C_VEL
LIN {X 0,Y 356.184,Z 340.164,A -85,B 0,C 180,E1 -13513.696,E2 -13513.696} C_VEL
LIN {X 0,Y 355.302,Z 346.173,A -85,B 0,C 180,E1 -13515.487,E2 -13515.487} C_VEL
LIN {X 0,Y 354.612,Z 350.816,A -85,B 0,C 180,E1 -13517.294,E2 -13517.294} C_VEL
LIN {X 0,Y 354.231,Z 353.249,A -85,B 0,C 180,E1 -13518.508,E2 -13518.508} C_VEL
LIN {X 0,Y 353.896,Z 355.204,A -85,B 0,C 180,E1 -13519.73,E2 -13519.73} C_VEL
LIN {X 0,Y 353.669,Z 356.604,A -85,B 0,C 180,E1 -13520.958,E2 -13520.958} C_VEL
LIN {X 0,Y 353.455,Z 357.558,A -85,B 0,C 180,E1 -13522.196,E2 -13522.196} C_VEL
LIN {X 0,Y 353.325,Z 358.027,A -85,B 0,C 180,E1 -13523.795,E2 -13523.795} C_VEL
LIN {X 0,Y 353.265,Z 357.401,A -85,B 0,C 180,E1 -13525.955,E2 -13525.955} C_VEL
LIN {X 0,Y 353.262,Z 356.292,A -85,B 0,C 180,E1 -13527.23,E2 -13527.23} C_VEL
LIN {X 0,Y 353.476,Z 353.932,A -85,B 0,C 180,E1 -13528.974,E2 -13528.974} C_VEL
LIN {X 0,Y 353.798,Z 349.651,A -85,B 0,C 180,E1 -13531.096,E2 -13531.096} C_VEL
LIN {X 0,Y 354.165,Z 344.306,A -85,B 0,C 180,E1 -13532.998,E2 -13532.998} C_VEL
LIN {X 0,Y 354.678,Z 338.05,A -85,B 0,C 180,E1 -13534.728,E2 -13534.728} C_VEL
LIN {X 0,Y 355.31,Z 330.531,A -85,B 0,C 180,E1 -13536.398,E2 -13536.398} C_VEL
LIN {X 0,Y 356.062,Z 321.295,A -85,B 0,C 180,E1 -13538.047,E2 -13538.047} C_VEL
LIN {X 0,Y 356.899,Z 311.06,A -85,B 0,C 180,E1 -13539.513,E2 -13539.513} C_VEL
LIN {X 0,Y 357.736,Z 300.029,A -85,B 0,C 180,E1 -13540.784,E2 -13540.784} C_VEL
LIN {X 0,Y 358.465,Z 288.447,A -85,B 0,C 180,E1 -13541.839,E2 -13541.839} C_VEL
LIN {X 0,Y 359.192,Z 276.338,A -85,B 0,C 180,E1 -13542.694,E2 -13542.694} C_VEL
LIN {X 0,Y 359.723,Z 263.241,A -85,B 0,C 180,E1 -13543.373,E2 -13543.373} C_VEL
LIN {X 0,Y 360.143,Z 249.733,A -85,B 0,C 180,E1 -13543.829,E2 -13543.829} C_VEL
LIN {X 0,Y 361.987,Z 169.715,A -85,B 0,C 180,E1 -13545.701,E2 -13545.701} C_VEL
LIN {X 0,Y 359.87,Z 160.803,A -85,B 0,C 180,E1 -13546.023,E2 -13546.023} C_VEL
LIN {X 0,Y 355.276,Z 146.363,A -85,B 0,C 180,E1 -13546.629,E2 -13546.629} C_VEL
LIN {X 0,Y 354.855,Z 144.285,A -85,B 0,C 180,E1 -13547.212,E2 -13547.212} C_VEL
LIN {X 0,Y 354.815,Z 144.284,A -85,B 0,C 180,E1 -13550.666,E2 -13550.666} C_VEL
LIN {X 0,Y 354.821,Z 144.284,A -85,B 0,C 180,E1 -13554.3,E2 -13554.3} C_VEL
LIN {X 0,Y 354.786,Z 144.292,A -85,B 0,C 180,E1 -13557.666,E2 -13557.666} C_VEL
LIN {X 0,Y 354.868,Z 144.278,A -85,B 0,C 180,E1 -13560.621,E2 -13560.621} C_VEL
LIN {X 0,Y 354.899,Z 144.274,A -85,B 0,C 180,E1 -13564.172,E2 -13564.172} C_VEL
LIN {X 0,Y 354.834,Z 144.283,A -85,B 0,C 180,E1 -13567.894,E2 -13567.894} C_VEL
LIN {X 0,Y 354.888,Z 144.276,A -85,B 0,C 180,E1 -13571.907,E2 -13571.907} C_VEL
LIN {X 0,Y 354.941,Z 144.269,A -85,B 0,C 180,E1 -13575.981,E2 -13575.981} C_VEL
LIN {X 0,Y 354.977,Z 144.265,A -85,B 0,C 180,E1 -13579.735,E2 -13579.735} C_VEL
LIN {X 0,Y 355.124,Z 144.25,A -85,B 0,C 180,E1 -13583.18,E2 -13583.18} C_VEL
LIN {X 0,Y 355.244,Z 144.231,A -85,B 0,C 180,E1 -13587.732,E2 -13587.732} C_VEL
LIN {X 0,Y 355.396,Z 144.212,A -85,B 0,C 180,E1 -13590,E2 -13590} C_VEL
LIN {X 0,Y 355.244,Z 144.232,A -85,B 0,C 180,E1 -13592.267,E2 -13592.267} C_VEL
LIN {X 0,Y 355.123,Z 144.25,A -85,B 0,C 180,E1 -13596.819,E2 -13596.819} C_VEL
LIN {X 0,Y 354.976,Z 144.267,A -85,B 0,C 180,E1 -13600.264,E2 -13600.264} C_VEL
LIN {X 0,Y 354.94,Z 144.27,A -85,B 0,C 180,E1 -13604.019,E2 -13604.019} C_VEL
LIN {X 0,Y 354.889,Z 144.275,A -85,B 0,C 180,E1 -13607.174,E2 -13607.174} C_VEL
LIN {X 0,Y 354.255,Z 144.359,A -85,B 0,C 180,E1 -13608.121,E2 -13608.121} C_VEL
LIN {X 0,Y 351.364,Z 144.716,A -85,B 0,C 180,E1 -13609.66,E2 -13609.66} C_VEL
LIN {X 0,Y 348.891,Z 145.024,A -85,B 0,C 180,E1 -13610.905,E2 -13610.905} C_VEL
LIN {X 0,Y 347.833,Z 145.156,A -85,B 0,C 180,E1 -13611.87,E2 -13611.87} C_VEL
LIN {X 0,Y 347.751,Z 145.165,A -85,B 0,C 180,E1 -13612.197,E2 -13612.197} C_VEL
LIN {X 0,Y 347.808,Z 145.157,A -85,B 0,C 180,E1 -13615.108,E2 -13615.108} C_VEL
LIN {X 0,Y 347.809,Z 145.158,A -85,B 0,C 180,E1 -13617.693,E2 -13617.693} C_VEL
LIN {X 0,Y 347.767,Z 145.166,A -85,B 0,C 180,E1 -13620.346,E2 -13620.346} C_VEL
LIN {X 0,Y 347.745,Z 145.171,A -85,B 0,C 180,E1 -13624.044,E2 -13624.044} C_VEL
LIN {X 0,Y 347.759,Z 145.164,A -85,B 0,C 180,E1 -13627.32,E2 -13627.32} C_VEL
LIN {X 0,Y 347.79,Z 145.162,A -85,B 0,C 180,E1 -13630.288,E2 -13630.288} C_VEL
LIN {X 0,Y 347.783,Z 145.162,A -85,B 0,C 180,E1 -13633.398,E2 -13633.398} C_VEL
LIN {X 0,Y 347.766,Z 145.163,A -85,B 0,C 180,E1 -13636.679,E2 -13636.679} C_VEL
LIN {X 0,Y 347.754,Z 145.166,A -85,B 0,C 180,E1 -13640.171,E2 -13640.171} C_VEL
LIN {X 0,Y 347.768,Z 145.165,A -85,B 0,C 180,E1 -13643.935,E2 -13643.935} C_VEL
LIN {X 0,Y 347.739,Z 145.166,A -85,B 0,C 180,E1 -13646.929,E2 -13646.929} C_VEL
LIN {X 0,Y 347.801,Z 145.159,A -85,B 0,C 180,E1 -13650.99,E2 -13650.99} C_VEL
LIN {X 0,Y 347.829,Z 145.159,A -85,B 0,C 180,E1 -13653.608,E2 -13653.608} C_VEL
LIN {X 0,Y 347.785,Z 145.16,A -85,B 0,C 180,E1 -13656.162,E2 -13656.162} C_VEL
LIN {X 0,Y 347.814,Z 145.157,A -85,B 0,C 180,E1 -13659.91,E2 -13659.91} C_VEL
LIN {X 0,Y 347.864,Z 145.15,A -85,B 0,C 180,E1 -13662.36,E2 -13662.36} C_VEL
LIN {X 0,Y 347.894,Z 145.147,A -85,B 0,C 180,E1 -13665.971,E2 -13665.971} C_VEL
LIN {X 0,Y 347.926,Z 145.145,A -85,B 0,C 180,E1 -13669.526,E2 -13669.526} C_VEL
LIN {X 0,Y 348.089,Z 145.128,A -85,B 0,C 180,E1 -13673.042,E2 -13673.042} C_VEL
LIN {X 0,Y 348.206,Z 145.108,A -85,B 0,C 180,E1 -13677.687,E2 -13677.687} C_VEL
LIN {X 0,Y 348.344,Z 145.09,A -85,B 0,C 180,E1 -13680,E2 -13680} C_VEL
LIN {X 0,Y 348.206,Z 145.109,A -85,B 0,C 180,E1 -13682.314,E2 -13682.314} C_VEL
LIN {X 0,Y 348.105,Z 145.124,A -85,B 0,C 180,E1 -13686.958,E2 -13686.958} C_VEL
LIN {X 0,Y 347.966,Z 145.138,A -85,B 0,C 180,E1 -13689.299,E2 -13689.299} C_VEL
LIN {X 0,Y 347.889,Z 145.151,A -85,B 0,C 180,E1 -13692.84,E2 -13692.84} C_VEL
LIN {X 0,Y 347.838,Z 145.159,A -85,B 0,C 180,E1 -13696.432,E2 -13696.432} C_VEL
LIN {X 0,Y 347.854,Z 145.154,A -85,B 0,C 180,E1 -13698.861,E2 -13698.861} C_VEL
LIN {X 0,Y 347.761,Z 145.167,A -85,B 0,C 180,E1 -13702.581,E2 -13702.581} C_VEL
LIN {X 0,Y 347.81,Z 145.157,A -85,B 0,C 180,E1 -13705.109,E2 -13705.109} C_VEL
LIN {X 0,Y 347.81,Z 145.158,A -85,B 0,C 180,E1 -13707.694,E2 -13707.694} C_VEL
LIN {X 0,Y 347.763,Z 145.168,A -85,B 0,C 180,E1 -13710.347,E2 -13710.347} C_VEL
LIN {X 0,Y 347.744,Z 145.168,A -85,B 0,C 180,E1 -13714.464,E2 -13714.464} C_VEL
LIN {X 0,Y 347.776,Z 145.167,A -85,B 0,C 180,E1 -13717.99,E2 -13717.99} C_VEL
LIN {X 0,Y 347.766,Z 145.167,A -85,B 0,C 180,E1 -13721.828,E2 -13721.828} C_VEL
LIN {X 0,Y 347.708,Z 145.17,A -85,B 0,C 180,E1 -13725.027,E2 -13725.027} C_VEL
LIN {X 0,Y 347.75,Z 145.166,A -85,B 0,C 180,E1 -13728.398,E2 -13728.398} C_VEL
LIN {X 0,Y 347.774,Z 145.165,A -85,B 0,C 180,E1 -13732.012,E2 -13732.012} C_VEL
LIN {X 0,Y 347.745,Z 145.17,A -85,B 0,C 180,E1 -13735.537,E2 -13735.537} C_VEL
LIN {X 0,Y 347.835,Z 145.305,A -85,B 0,C 180,E1 -13739.114,E2 -13739.114} C_VEL
LIN {X 0,Y 350.756,Z 159.323,A -85,B 0,C 180,E1 -13742.559,E2 -13742.559} C_VEL
LIN {X 0,Y 351.645,Z 165.066,A -85,B 0,C 180,E1 -13743.916,E2 -13743.916} C_VEL
LIN {X 0,Y 350.099,Z 181.664,A -85,B 0,C 180,E1 -13747.579,E2 -13747.579} C_VEL
LIN {X 0,Y 349.911,Z 184.076,A -85,B 0,C 180,E1 -13748.11,E2 -13748.11} C_VEL
LIN {X 0,Y 354.458,Z 222.465,A -85,B 0,C 180,E1 -13749.305,E2 -13749.305} C_VEL
LIN {X 0,Y 352.875,Z 293.485,A -85,B 0,C 180,E1 -13751.042,E2 -13751.042} C_VEL
LIN {X 0,Y 352.176,Z 307.235,A -85,B 0,C 180,E1 -13751.606,E2 -13751.606} C_VEL
LIN {X 0,Y 351.39,Z 319.248,A -85,B 0,C 180,E1 -13752.317,E2 -13752.317} C_VEL
LIN {X 0,Y 350.426,Z 331.004,A -85,B 0,C 180,E1 -13753.244,E2 -13753.244} C_VEL
LIN {X 0,Y 349.46,Z 342.445,A -85,B 0,C 180,E1 -13754.397,E2 -13754.397} C_VEL
LIN {X 0,Y 348.535,Z 353.218,A -85,B 0,C 180,E1 -13755.76,E2 -13755.76} C_VEL
LIN {X 0,Y 347.817,Z 362.143,A -85,B 0,C 180,E1 -13757.158,E2 -13757.158} C_VEL
LIN {X 0,Y 347.205,Z 369.837,A -85,B 0,C 180,E1 -13758.618,E2 -13758.618} C_VEL
LIN {X 0,Y 346.716,Z 377.376,A -85,B 0,C 180,E1 -13760.374,E2 -13760.374} C_VEL
LIN {X 0,Y 346.493,Z 382.462,A -85,B 0,C 180,E1 -13761.838,E2 -13761.838} C_VEL
LIN {X 0,Y 346.298,Z 387.357,A -85,B 0,C 180,E1 -13763.592,E2 -13763.592} C_VEL
LIN {X 0,Y 346.341,Z 391.065,A -85,B 0,C 180,E1 -13765.345,E2 -13765.345} C_VEL
LIN {X 0,Y 346.255,Z 392.936,A -85,B 0,C 180,E1 -13766.509,E2 -13766.509} C_VEL
LIN {X 0,Y 346.35,Z 394.318,A -85,B 0,C 180,E1 -13767.675,E2 -13767.675} C_VEL
LIN {X 0,Y 346.412,Z 395.272,A -85,B 0,C 180,E1 -13768.838,E2 -13768.838} C_VEL
LIN {X 0,Y 346.398,Z 395.803,A -85,B 0,C 180,E1 -13770,E2 -13770} C_VEL
LIN {X 0,Y 346.35,Z 395.882,A -85,B 0,C 180,E1 -13771.163,E2 -13771.163} C_VEL
LIN {X 0,Y 346.233,Z 395.515,A -85,B 0,C 180,E1 -13772.327,E2 -13772.327} C_VEL
LIN {X 0,Y 346.201,Z 394.742,A -85,B 0,C 180,E1 -13773.492,E2 -13773.492} C_VEL
LIN {X 0,Y 346.198,Z 393.557,A -85,B 0,C 180,E1 -13774.658,E2 -13774.658} C_VEL
LIN {X 0,Y 346.212,Z 390.919,A -85,B 0,C 180,E1 -13776.411,E2 -13776.411} C_VEL
LIN {X 0,Y 346.481,Z 387.259,A -85,B 0,C 180,E1 -13778.163,E2 -13778.163} C_VEL
LIN {X 0,Y 346.875,Z 382.491,A -85,B 0,C 180,E1 -13779.917,E2 -13779.917} C_VEL
LIN {X 0,Y 347.524,Z 376.48,A -85,B 0,C 180,E1 -13781.668,E2 -13781.668} C_VEL
LIN {X 0,Y 348.572,Z 368.986,A -85,B 0,C 180,E1 -13783.407,E2 -13783.407} C_VEL
LIN {X 0,Y 349.697,Z 359.736,A -85,B 0,C 180,E1 -13785.146,E2 -13785.146} C_VEL
LIN {X 0,Y 351.028,Z 350.277,A -85,B 0,C 180,E1 -13786.577,E2 -13786.577} C_VEL
LIN {X 0,Y 352.664,Z 338.57,A -85,B 0,C 180,E1 -13787.993,E2 -13787.993} C_VEL
LIN {X 0,Y 354.216,Z 326.897,A -85,B 0,C 180,E1 -13789.11,E2 -13789.11} C_VEL
LIN {X 0,Y 355.438,Z 314.72,A -85,B 0,C 180,E1 -13790.018,E2 -13790.018} C_VEL
LIN {X 0,Y 356.823,Z 300.886,A -85,B 0,C 180,E1 -13790.765,E2 -13790.765} C_VEL
LIN {X 0,Y 357.615,Z 287.747,A -85,B 0,C 180,E1 -13791.244,E2 -13791.244} C_VEL
LIN {X 0,Y 359.821,Z 222.511,A -85,B 0,C 180,E1 -13792.913,E2 -13792.913} C_VEL
LIN {X 0,Y 357.994,Z 207.298,A -85,B 0,C 180,E1 -13793.537,E2 -13793.537} C_VEL
LIN {X 0,Y 354.992,Z 190.713,A -85,B 0,C 180,E1 -13794.332,E2 -13794.332} C_VEL
LIN {X 0,Y 352.598,Z 179.646,A -85,B 0,C 180,E1 -13794.941,E2 -13794.941} C_VEL
LIN {X 0,Y 353.627,Z 171.672,A -85,B 0,C 180,E1 -13796.741,E2 -13796.741} C_VEL
LIN {X 0,Y 353.448,Z 168.451,A -85,B 0,C 180,E1 -13797.536,E2 -13797.536} C_VEL
LIN {X 0,Y 351.571,Z 159.399,A -85,B 0,C 180,E1 -13799.984,E2 -13799.984} C_VEL
LIN {X 0,Y 349.483,Z 151.226,A -85,B 0,C 180,E1 -13802.369,E2 -13802.369} C_VEL
LIN {X 0,Y 347.769,Z 145.166,A -85,B 0,C 180,E1 -13804.331,E2 -13804.331} C_VEL
LIN {X 0,Y 347.778,Z 145.167,A -85,B 0,C 180,E1 -13807.989,E2 -13807.989} C_VEL
LIN {X 0,Y 347.754,Z 145.167,A -85,B 0,C 180,E1 -13811.83,E2 -13811.83} C_VEL
LIN {X 0,Y 347.709,Z 145.173,A -85,B 0,C 180,E1 -13815.027,E2 -13815.027} C_VEL
LIN {X 0,Y 347.754,Z 145.161,A -85,B 0,C 180,E1 -13818.397,E2 -13818.397} C_VEL
LIN {X 0,Y 347.776,Z 145.162,A -85,B 0,C 180,E1 -13822.011,E2 -13822.011} C_VEL
LIN {X 0,Y 347.748,Z 145.162,A -85,B 0,C 180,E1 -13825.536,E2 -13825.536} C_VEL
LIN {X 0,Y 347.748,Z 145.161,A -85,B 0,C 180,E1 -13828.3,E2 -13828.3} C_VEL
LIN {X 0,Y 347.782,Z 145.161,A -85,B 0,C 180,E1 -13830.987,E2 -13830.987} C_VEL
LIN {X 0,Y 347.834,Z 145.153,A -85,B 0,C 180,E1 -13833.608,E2 -13833.608} C_VEL
LIN {X 0,Y 347.792,Z 145.161,A -85,B 0,C 180,E1 -13836.162,E2 -13836.162} C_VEL
LIN {X 0,Y 347.815,Z 145.155,A -85,B 0,C 180,E1 -13839.909,E2 -13839.909} C_VEL
LIN {X 0,Y 347.835,Z 145.156,A -85,B 0,C 180,E1 -13843.568,E2 -13843.568} C_VEL
LIN {X 0,Y 347.893,Z 145.149,A -85,B 0,C 180,E1 -13847.16,E2 -13847.16} C_VEL
LIN {X 0,Y 347.938,Z 145.144,A -85,B 0,C 180,E1 -13850.7,E2 -13850.7} C_VEL
LIN {X 0,Y 348.071,Z 145.132,A -85,B 0,C 180,E1 -13853.041,E2 -13853.041} C_VEL
LIN {X 0,Y 348.196,Z 145.288,A -85,B 0,C 180,E1 -13857.975,E2 -13857.975} C_VEL
LIN {X 0,Y 349.85,Z 150.992,A -85,B 0,C 180,E1 -13859.838,E2 -13859.838} C_VEL
LIN {X 0,Y 356.439,Z 164.419,A -85,B 0,C 180,E1 -13860.984,E2 -13860.984} C_VEL
LIN {X 0,Y 361.322,Z 175.793,A -85,B 0,C 180,E1 -13861.818,E2 -13861.818} C_VEL
LIN {X 0,Y 358.176,Z 258.476,A -85,B 0,C 180,E1 -13863.973,E2 -13863.973} C_VEL
LIN {X 0,Y 357.45,Z 272.337,A -85,B 0,C 180,E1 -13864.581,E2 -13864.581} C_VEL
LIN {X 0,Y 356.506,Z 284.853,A -85,B 0,C 180,E1 -13865.373,E2 -13865.373} C_VEL
LIN {X 0,Y 355.307,Z 297.02,A -85,B 0,C 180,E1 -13866.388,E2 -13866.388} C_VEL
LIN {X 0,Y 354.057,Z 307.818,A -85,B 0,C 180,E1 -13867.536,E2 -13867.536} C_VEL
LIN {X 0,Y 352.725,Z 317.921,A -85,B 0,C 180,E1 -13868.883,E2 -13868.883} C_VEL
LIN {X 0,Y 351.429,Z 326.976,A -85,B 0,C 180,E1 -13870.368,E2 -13870.368} C_VEL
LIN {X 0,Y 350.311,Z 334.461,A -85,B 0,C 180,E1 -13871.866,E2 -13871.866} C_VEL
LIN {X 0,Y 349.161,Z 341.745,A -85,B 0,C 180,E1 -13873.68,E2 -13873.68} C_VEL
LIN {X 0,Y 348.388,Z 346.649,A -85,B 0,C 180,E1 -13875.203,E2 -13875.203} C_VEL
LIN {X 0,Y 347.632,Z 351.287,A -85,B 0,C 180,E1 -13877.046,E2 -13877.046} C_VEL
LIN {X 0,Y 347.036,Z 354.727,A -85,B 0,C 180,E1 -13878.906,E2 -13878.906} C_VEL
LIN {X 0,Y 346.553,Z 357.336,A -85,B 0,C 180,E1 -13881.113,E2 -13881.113} C_VEL
LIN {X 0,Y 346.304,Z 358.245,A -85,B 0,C 180,E1 -13882.68,E2 -13882.68} C_VEL
LIN {X 0,Y 346.234,Z 358.457,A -85,B 0,C 180,E1 -13884.016,E2 -13884.016} C_VEL
LIN {X 0,Y 346.169,Z 358.129,A -85,B 0,C 180,E1 -13885.235,E2 -13885.235} C_VEL
LIN {X 0,Y 346.17,Z 357.161,A -85,B 0,C 180,E1 -13886.709,E2 -13886.709} C_VEL
LIN {X 0,Y 346.217,Z 355.946,A -85,B 0,C 180,E1 -13887.832,E2 -13887.832} C_VEL
LIN {X 0,Y 346.521,Z 352.807,A -85,B 0,C 180,E1 -13889.811,E2 -13889.811} C_VEL
LIN {X 0,Y 346.839,Z 348.318,A -85,B 0,C 180,E1 -13891.792,E2 -13891.792} C_VEL
LIN {X 0,Y 347.233,Z 343.086,A -85,B 0,C 180,E1 -13893.543,E2 -13893.543} C_VEL
LIN {X 0,Y 347.717,Z 336.999,A -85,B 0,C 180,E1 -13895.172,E2 -13895.172} C_VEL
LIN {X 0,Y 348.445,Z 328.982,A -85,B 0,C 180,E1 -13896.895,E2 -13896.895} C_VEL
LIN {X 0,Y 349.265,Z 319.156,A -85,B 0,C 180,E1 -13898.593,E2 -13898.593} C_VEL
LIN {X 0,Y 350.102,Z 309.256,A -85,B 0,C 180,E1 -13899.968,E2 -13899.968} C_VEL
LIN {X 0,Y 350.907,Z 298.242,A -85,B 0,C 180,E1 -13901.201,E2 -13901.201} C_VEL
LIN {X 0,Y 351.695,Z 286.449,A -85,B 0,C 180,E1 -13902.25,E2 -13902.25} C_VEL
LIN {X 0,Y 352.428,Z 274.232,A -85,B 0,C 180,E1 -13903.078,E2 -13903.078} C_VEL
LIN {X 0,Y 352.863,Z 261.789,A -85,B 0,C 180,E1 -13903.699,E2 -13903.699} C_VEL
LIN {X 0,Y 353.275,Z 248.606,A -85,B 0,C 180,E1 -13904.129,E2 -13904.129} C_VEL
LIN {X 0,Y 355.185,Z 170.729,A -85,B 0,C 180,E1 -13905.991,E2 -13905.991} C_VEL
LIN {X 0,Y 353.158,Z 162.489,A -85,B 0,C 180,E1 -13906.297,E2 -13906.297} C_VEL
LIN {X 0,Y 348.106,Z 146.733,A -85,B 0,C 180,E1 -13906.973,E2 -13906.973} C_VEL
LIN {X 0,Y 347.797,Z 145.164,A -85,B 0,C 180,E1 -13907.444,E2 -13907.444} C_VEL
LIN {X 0,Y 347.751,Z 145.166,A -85,B 0,C 180,E1 -13911.207,E2 -13911.207} C_VEL
LIN {X 0,Y 347.788,Z 145.161,A -85,B 0,C 180,E1 -13914.124,E2 -13914.124} C_VEL
LIN {X 0,Y 347.737,Z 145.167,A -85,B 0,C 180,E1 -13918.086,E2 -13918.086} C_VEL
LIN {X 0,Y 347.804,Z 145.16,A -85,B 0,C 180,E1 -13920.99,E2 -13920.99} C_VEL
LIN {X 0,Y 347.831,Z 145.158,A -85,B 0,C 180,E1 -13923.607,E2 -13923.607} C_VEL
LIN {X 0,Y 347.788,Z 145.16,A -85,B 0,C 180,E1 -13926.161,E2 -13926.161} C_VEL
LIN {X 0,Y 347.804,Z 145.158,A -85,B 0,C 180,E1 -13929.908,E2 -13929.908} C_VEL
LIN {X 0,Y 347.831,Z 145.157,A -85,B 0,C 180,E1 -13933.568,E2 -13933.568} C_VEL
LIN {X 0,Y 347.889,Z 145.153,A -85,B 0,C 180,E1 -13937.16,E2 -13937.16} C_VEL
LIN {X 0,Y 347.963,Z 145.141,A -85,B 0,C 180,E1 -13940.701,E2 -13940.701} C_VEL
LIN {X 0,Y 348.09,Z 145.127,A -85,B 0,C 180,E1 -13943.042,E2 -13943.042} C_VEL
LIN {X 0,Y 348.207,Z 145.108,A -85,B 0,C 180,E1 -13947.686,E2 -13947.686} C_VEL
LIN {X 0,Y 348.345,Z 145.09,A -85,B 0,C 180,E1 -13950,E2 -13950} C_VEL
LIN {X 0,Y 348.206,Z 145.109,A -85,B 0,C 180,E1 -13952.313,E2 -13952.313} C_VEL
LIN {X 0,Y 348.09,Z 145.125,A -85,B 0,C 180,E1 -13956.958,E2 -13956.958} C_VEL
LIN {X 0,Y 347.927,Z 145.147,A -85,B 0,C 180,E1 -13960.474,E2 -13960.474} C_VEL
LIN {X 0,Y 347.896,Z 145.149,A -85,B 0,C 180,E1 -13964.149,E2 -13964.149} C_VEL
LIN {X 0,Y 347.889,Z 145.152,A -85,B 0,C 180,E1 -13968.29,E2 -13968.29} C_VEL
LIN {X 0,Y 347.751,Z 145.165,A -85,B 0,C 180,E1 -13972.197,E2 -13972.197} C_VEL
LIN {X 0,Y 347.106,Z 145.248,A -85,B 0,C 180,E1 -13973.164,E2 -13973.164} C_VEL
LIN {X 0,Y 344.304,Z 145.597,A -85,B 0,C 180,E1 -13974.739,E2 -13974.739} C_VEL
LIN {X 0,Y 341.913,Z 145.895,A -85,B 0,C 180,E1 -13976.013,E2 -13976.013} C_VEL
LIN {X 0,Y 340.874,Z 146.022,A -85,B 0,C 180,E1 -13976.999,E2 -13976.999} C_VEL
LIN {X 0,Y 340.782,Z 146.032,A -85,B 0,C 180,E1 -13977.332,E2 -13977.332} C_VEL
LIN {X 0,Y 340.762,Z 146.039,A -85,B 0,C 180,E1 -13979.978,E2 -13979.978} C_VEL
LIN {X 0,Y 340.692,Z 146.047,A -85,B 0,C 180,E1 -13983.846,E2 -13983.846} C_VEL
LIN {X 0,Y 340.702,Z 146.043,A -85,B 0,C 180,E1 -13986.741,E2 -13986.741} C_VEL
LIN {X 0,Y 340.76,Z 146.038,A -85,B 0,C 180,E1 -13990.262,E2 -13990.262} C_VEL
LIN {X 0,Y 340.732,Z 146.044,A -85,B 0,C 180,E1 -13993.788,E2 -13993.788} C_VEL
LIN {X 0,Y 340.73,Z 146.043,A -85,B 0,C 180,E1 -13997.948,E2 -13997.948} C_VEL
LIN {X 0,Y 340.735,Z 146.044,A -85,B 0,C 180,E1 -14001.774,E2 -14001.774} C_VEL
LIN {X 0,Y 340.719,Z 146.046,A -85,B 0,C 180,E1 -14005.595,E2 -14005.595} C_VEL
LIN {X 0,Y 340.701,Z 146.044,A -85,B 0,C 180,E1 -14008.956,E2 -14008.956} C_VEL
LIN {X 0,Y 340.775,Z 146.033,A -85,B 0,C 180,E1 -14012.474,E2 -14012.474} C_VEL
LIN {X 0,Y 340.753,Z 146.04,A -85,B 0,C 180,E1 -14015.639,E2 -14015.639} C_VEL
LIN {X 0,Y 340.746,Z 146.041,A -85,B 0,C 180,E1 -14019.475,E2 -14019.475} C_VEL
LIN {X 0,Y 340.855,Z 146.024,A -85,B 0,C 180,E1 -14021.985,E2 -14021.985} C_VEL
LIN {X 0,Y 340.866,Z 146.023,A -85,B 0,C 180,E1 -14025.705,E2 -14025.705} C_VEL
LIN {X 0,Y 340.868,Z 146.026,A -85,B 0,C 180,E1 -14029.307,E2 -14029.307} C_VEL
LIN {X 0,Y 341.057,Z 146.003,A -85,B 0,C 180,E1 -14032.898,E2 -14032.898} C_VEL
LIN {X 0,Y 341.168,Z 145.985,A -85,B 0,C 180,E1 -14037.639,E2 -14037.639} C_VEL
LIN {X 0,Y 341.295,Z 145.969,A -85,B 0,C 180,E1 -14040,E2 -14040} C_VEL
LIN {X 0,Y 341.168,Z 145.986,A -85,B 0,C 180,E1 -14042.362,E2 -14042.362} C_VEL
LIN {X 0,Y 341.074,Z 145.998,A -85,B 0,C 180,E1 -14047.102,E2 -14047.102} C_VEL
LIN {X 0,Y 340.869,Z 146.027,A -85,B 0,C 180,E1 -14050.694,E2 -14050.694} C_VEL
LIN {X 0,Y 340.861,Z 146.026,A -85,B 0,C 180,E1 -14054.325,E2 -14054.325} C_VEL
LIN {X 0,Y 340.837,Z 146.032,A -85,B 0,C 180,E1 -14058.467,E2 -14058.467} C_VEL
LIN {X 0,Y 340.716,Z 146.042,A -85,B 0,C 180,E1 -14061.842,E2 -14061.842} C_VEL
LIN {X 0,Y 340.771,Z 146.035,A -85,B 0,C 180,E1 -14065.665,E2 -14065.665} C_VEL
LIN {X 0,Y 340.74,Z 146.043,A -85,B 0,C 180,E1 -14068.32,E2 -14068.32} C_VEL
LIN {X 0,Y 340.703,Z 146.042,A -85,B 0,C 180,E1 -14071.045,E2 -14071.045} C_VEL
LIN {X 0,Y 340.718,Z 146.041,A -85,B 0,C 180,E1 -14075.279,E2 -14075.279} C_VEL
LIN {X 0,Y 340.717,Z 146.043,A -85,B 0,C 180,E1 -14078.388,E2 -14078.388} C_VEL
LIN {X 0,Y 340.731,Z 146.044,A -85,B 0,C 180,E1 -14082.052,E2 -14082.052} C_VEL
LIN {X 0,Y 340.652,Z 146.051,A -85,B 0,C 180,E1 -14086.227,E2 -14086.227} C_VEL
LIN {X 0,Y 340.689,Z 146.05,A -85,B 0,C 180,E1 -14089.754,E2 -14089.754} C_VEL
LIN {X 0,Y 340.705,Z 146.044,A -85,B 0,C 180,E1 -14093.259,E2 -14093.259} C_VEL
LIN {X 0,Y 340.693,Z 146.045,A -85,B 0,C 180,E1 -14096.154,E2 -14096.154} C_VEL
LIN {X 0,Y 340.738,Z 146.103,A -85,B 0,C 180,E1 -14098.831,E2 -14098.831} C_VEL
LIN {X 0,Y 343.639,Z 159.814,A -85,B 0,C 180,E1 -14102.272,E2 -14102.272} C_VEL
LIN {X 0,Y 344.655,Z 166.111,A -85,B 0,C 180,E1 -14103.796,E2 -14103.796} C_VEL
LIN {X 0,Y 342.965,Z 183.666,A -85,B 0,C 180,E1 -14107.748,E2 -14107.748} C_VEL
LIN {X 0,Y 347.606,Z 223.549,A -85,B 0,C 180,E1 -14109.035,E2 -14109.035} C_VEL
LIN {X 0,Y 345.969,Z 292.776,A -85,B 0,C 180,E1 -14110.764,E2 -14110.764} C_VEL
LIN {X 0,Y 345.274,Z 306.609,A -85,B 0,C 180,E1 -14111.34,E2 -14111.34} C_VEL
LIN {X 0,Y 344.431,Z 319.196,A -85,B 0,C 180,E1 -14112.101,E2 -14112.101} C_VEL
LIN {X 0,Y 343.444,Z 330.878,A -85,B 0,C 180,E1 -14113.047,E2 -14113.047} C_VEL
LIN {X 0,Y 342.455,Z 342.275,A -85,B 0,C 180,E1 -14114.222,E2 -14114.222} C_VEL
LIN {X 0,Y 341.512,Z 352.567,A -85,B 0,C 180,E1 -14115.547,E2 -14115.547} C_VEL
LIN {X 0,Y 340.823,Z 361.066,A -85,B 0,C 180,E1 -14116.89,E2 -14116.89} C_VEL
LIN {X 0,Y 340.211,Z 368.883,A -85,B 0,C 180,E1 -14118.381,E2 -14118.381} C_VEL
LIN {X 0,Y 339.656,Z 376.521,A -85,B 0,C 180,E1 -14120.172,E2 -14120.172} C_VEL
LIN {X 0,Y 339.429,Z 381.699,A -85,B 0,C 180,E1 -14121.667,E2 -14121.667} C_VEL
LIN {X 0,Y 339.228,Z 386.677,A -85,B 0,C 180,E1 -14123.458,E2 -14123.458} C_VEL
LIN {X 0,Y 339.248,Z 390.459,A -85,B 0,C 180,E1 -14125.247,E2 -14125.247} C_VEL
LIN {X 0,Y 339.179,Z 392.378,A -85,B 0,C 180,E1 -14126.437,E2 -14126.437} C_VEL
LIN {X 0,Y 339.254,Z 393.812,A -85,B 0,C 180,E1 -14127.626,E2 -14127.626} C_VEL
LIN {X 0,Y 339.35,Z 394.799,A -85,B 0,C 180,E1 -14128.814,E2 -14128.814} C_VEL
LIN {X 0,Y 339.336,Z 395.36,A -85,B 0,C 180,E1 -14130,E2 -14130} C_VEL
LIN {X 0,Y 339.255,Z 395.49,A -85,B 0,C 180,E1 -14131.187,E2 -14131.187} C_VEL
LIN {X 0,Y 339.137,Z 395.152,A -85,B 0,C 180,E1 -14132.376,E2 -14132.376} C_VEL
LIN {X 0,Y 339.121,Z 394.409,A -85,B 0,C 180,E1 -14133.565,E2 -14133.565} C_VEL
LIN {X 0,Y 339.076,Z 391.904,A -85,B 0,C 180,E1 -14135.789,E2 -14135.789} C_VEL
LIN {X 0,Y 339.325,Z 388.424,A -85,B 0,C 180,E1 -14137.737,E2 -14137.737} C_VEL
LIN {X 0,Y 339.687,Z 384.099,A -85,B 0,C 180,E1 -14139.528,E2 -14139.528} C_VEL
LIN {X 0,Y 340.404,Z 377.517,A -85,B 0,C 180,E1 -14141.613,E2 -14141.613} C_VEL
LIN {X 0,Y 341.461,Z 370.399,A -85,B 0,C 180,E1 -14143.389,E2 -14143.389} C_VEL
LIN {X 0,Y 342.511,Z 362.298,A -85,B 0,C 180,E1 -14145.042,E2 -14145.042} C_VEL
LIN {X 0,Y 343.948,Z 352.673,A -85,B 0,C 180,E1 -14146.623,E2 -14146.623} C_VEL
LIN {X 0,Y 345.522,Z 341.753,A -85,B 0,C 180,E1 -14148.071,E2 -14148.071} C_VEL
LIN {X 0,Y 347.142,Z 330.926,A -85,B 0,C 180,E1 -14149.208,E2 -14149.208} C_VEL
LIN {X 0,Y 348.521,Z 319.023,A -85,B 0,C 180,E1 -14150.202,E2 -14150.202} C_VEL
LIN {X 0,Y 349.991,Z 305.676,A -85,B 0,C 180,E1 -14151.035,E2 -14151.035} C_VEL
LIN {X 0,Y 351.022,Z 292.115,A -85,B 0,C 180,E1 -14151.625,E2 -14151.625} C_VEL
LIN {X 0,Y 352.257,Z 262.776,A -85,B 0,C 180,E1 -14152.42,E2 -14152.42} C_VEL
LIN {X 0,Y 353.629,Z 222.955,A -85,B 0,C 180,E1 -14153.48,E2 -14153.48} C_VEL
LIN {X 0,Y 351.657,Z 206.968,A -85,B 0,C 180,E1 -14154.168,E2 -14154.168} C_VEL
LIN {X 0,Y 348.498,Z 190.066,A -85,B 0,C 180,E1 -14155.03,E2 -14155.03} C_VEL
LIN {X 0,Y 346.101,Z 179.051,A -85,B 0,C 180,E1 -14155.685,E2 -14155.685} C_VEL
LIN {X 0,Y 346.956,Z 172.411,A -85,B 0,C 180,E1 -14157.226,E2 -14157.226} C_VEL
LIN {X 0,Y 345.413,Z 163.836,A -85,B 0,C 180,E1 -14159.565,E2 -14159.565} C_VEL
LIN {X 0,Y 343.289,Z 155.052,A -85,B 0,C 180,E1 -14162.16,E2 -14162.16} C_VEL
LIN {X 0,Y 340.717,Z 146.045,A -85,B 0,C 180,E1 -14165.156,E2 -14165.156} C_VEL
LIN {X 0,Y 340.713,Z 146.045,A -85,B 0,C 180,E1 -14168.386,E2 -14168.386} C_VEL
LIN {X 0,Y 340.703,Z 146.044,A -85,B 0,C 180,E1 -14172.045,E2 -14172.045} C_VEL
LIN {X 0,Y 340.655,Z 146.048,A -85,B 0,C 180,E1 -14176.227,E2 -14176.227} C_VEL
LIN {X 0,Y 340.692,Z 146.046,A -85,B 0,C 180,E1 -14179.753,E2 -14179.753} C_VEL
LIN {X 0,Y 340.708,Z 146.037,A -85,B 0,C 180,E1 -14183.258,E2 -14183.258} C_VEL
LIN {X 0,Y 340.696,Z 146.038,A -85,B 0,C 180,E1 -14186.153,E2 -14186.153} C_VEL
LIN {X 0,Y 340.745,Z 146.039,A -85,B 0,C 180,E1 -14190.329,E2 -14190.329} C_VEL
LIN {X 0,Y 340.807,Z 146.035,A -85,B 0,C 180,E1 -14193.02,E2 -14193.02} C_VEL
LIN {X 0,Y 340.76,Z 146.039,A -85,B 0,C 180,E1 -14195.638,E2 -14195.638} C_VEL
LIN {X 0,Y 340.755,Z 146.034,A -85,B 0,C 180,E1 -14199.474,E2 -14199.474} C_VEL
LIN {X 0,Y 340.796,Z 146.028,A -85,B 0,C 180,E1 -14201.98,E2 -14201.98} C_VEL
LIN {X 0,Y 340.873,Z 146.025,A -85,B 0,C 180,E1 -14205.705,E2 -14205.705} C_VEL
LIN {X 0,Y 340.851,Z 146.027,A -85,B 0,C 180,E1 -14209.305,E2 -14209.305} C_VEL
LIN {X 0,Y 341.019,Z 146.009,A -85,B 0,C 180,E1 -14212.897,E2 -14212.897} C_VEL
LIN {X 0,Y 341.041,Z 146.125,A -85,B 0,C 180,E1 -14217.12,E2 -14217.12} C_VEL
LIN {X 0,Y 342.688,Z 151.569,A -85,B 0,C 180,E1 -14219.008,E2 -14219.008} C_VEL
LIN {X 0,Y 346.816,Z 159.285,A -85,B 0,C 180,E1 -14219.763,E2 -14219.763} C_VEL
LIN {X 0,Y 351.734,Z 169.608,A -85,B 0,C 180,E1 -14220.653,E2 -14220.653} C_VEL
LIN {X 0,Y 355.254,Z 178.015,A -85,B 0,C 180,E1 -14221.283,E2 -14221.283} C_VEL
LIN {X 0,Y 351.927,Z 258.727,A -85,B 0,C 180,E1 -14223.434,E2 -14223.434} C_VEL
LIN {X 0,Y 351.186,Z 271.851,A -85,B 0,C 180,E1 -14224.016,E2 -14224.016} C_VEL
LIN {X 0,Y 350.286,Z 283.592,A -85,B 0,C 180,E1 -14224.747,E2 -14224.747} C_VEL
LIN {X 0,Y 349.032,Z 296.098,A -85,B 0,C 180,E1 -14225.778,E2 -14225.778} C_VEL
LIN {X 0,Y 347.636,Z 307.394,A -85,B 0,C 180,E1 -14226.967,E2 -14226.967} C_VEL
LIN {X 0,Y 346.403,Z 316.535,A -85,B 0,C 180,E1 -14228.164,E2 -14228.164} C_VEL
LIN {X 0,Y 344.98,Z 325.913,A -85,B 0,C 180,E1 -14229.675,E2 -14229.675} C_VEL
LIN {X 0,Y 343.638,Z 334.429,A -85,B 0,C 180,E1 -14231.379,E2 -14231.379} C_VEL
LIN {X 0,Y 342.488,Z 341.153,A -85,B 0,C 180,E1 -14233.045,E2 -14233.045} C_VEL
LIN {X 0,Y 341.412,Z 347.515,A -85,B 0,C 180,E1 -14235.052,E2 -14235.052} C_VEL
LIN {X 0,Y 340.663,Z 351.756,A -85,B 0,C 180,E1 -14236.787,E2 -14236.787} C_VEL
LIN {X 0,Y 340.203,Z 354.334,A -85,B 0,C 180,E1 -14238.142,E2 -14238.142} C_VEL
LIN {X 0,Y 339.878,Z 356.091,A -85,B 0,C 180,E1 -14239.32,E2 -14239.32} C_VEL
LIN {X 0,Y 339.452,Z 358.047,A -85,B 0,C 180,E1 -14241.301,E2 -14241.301} C_VEL
LIN {X 0,Y 339.174,Z 358.831,A -85,B 0,C 180,E1 -14243.184,E2 -14243.184} C_VEL
LIN {X 0,Y 339.113,Z 358.752,A -85,B 0,C 180,E1 -14244.487,E2 -14244.487} C_VEL
LIN {X 0,Y 339.066,Z 358.195,A -85,B 0,C 180,E1 -14245.803,E2 -14245.803} C_VEL
LIN {X 0,Y 339.082,Z 357.067,A -85,B 0,C 180,E1 -14247.128,E2 -14247.128} C_VEL
LIN {X 0,Y 339.199,Z 355.443,A -85,B 0,C 180,E1 -14248.46,E2 -14248.46} C_VEL
LIN {X 0,Y 339.538,Z 351.878,A -85,B 0,C 180,E1 -14250.472,E2 -14250.472} C_VEL
LIN {X 0,Y 339.896,Z 346.797,A -85,B 0,C 180,E1 -14252.52,E2 -14252.52} C_VEL
LIN {X 0,Y 340.393,Z 340.983,A -85,B 0,C 180,E1 -14254.323,E2 -14254.323} C_VEL
LIN {X 0,Y 340.958,Z 334.348,A -85,B 0,C 180,E1 -14255.976,E2 -14255.976} C_VEL
LIN {X 0,Y 341.707,Z 325.644,A -85,B 0,C 180,E1 -14257.725,E2 -14257.725} C_VEL
LIN {X 0,Y 342.513,Z 316.143,A -85,B 0,C 180,E1 -14259.266,E2 -14259.266} C_VEL
LIN {X 0,Y 343.303,Z 306.867,A -85,B 0,C 180,E1 -14260.498,E2 -14260.498} C_VEL
LIN {X 0,Y 344.229,Z 295.023,A -85,B 0,C 180,E1 -14261.766,E2 -14261.766} C_VEL
LIN {X 0,Y 345.002,Z 283.241,A -85,B 0,C 180,E1 -14262.752,E2 -14262.752} C_VEL
LIN {X 0,Y 345.684,Z 270.195,A -85,B 0,C 180,E1 -14263.58,E2 -14263.58} C_VEL
LIN {X 0,Y 346.178,Z 256.379,A -85,B 0,C 180,E1 -14264.18,E2 -14264.18} C_VEL
LIN {X 0,Y 347.208,Z 215.187,A -85,B 0,C 180,E1 -14265.219,E2 -14265.219} C_VEL
LIN {X 0,Y 348.285,Z 171.245,A -85,B 0,C 180,E1 -14266.305,E2 -14266.305} C_VEL
LIN {X 0,Y 345.613,Z 161.482,A -85,B 0,C 180,E1 -14266.693,E2 -14266.693} C_VEL
LIN {X 0,Y 340.989,Z 147.132,A -85,B 0,C 180,E1 -14267.321,E2 -14267.321} C_VEL
LIN {X 0,Y 340.748,Z 146.043,A -85,B 0,C 180,E1 -14267.708,E2 -14267.708} C_VEL
LIN {X 0,Y 340.732,Z 146.043,A -85,B 0,C 180,E1 -14271.772,E2 -14271.772} C_VEL
LIN {X 0,Y 340.722,Z 146.046,A -85,B 0,C 180,E1 -14275.595,E2 -14275.595} C_VEL
LIN {X 0,Y 340.703,Z 146.044,A -85,B 0,C 180,E1 -14278.955,E2 -14278.955} C_VEL
LIN {X 0,Y 340.778,Z 146.033,A -85,B 0,C 180,E1 -14282.474,E2 -14282.474} C_VEL
LIN {X 0,Y 340.755,Z 146.039,A -85,B 0,C 180,E1 -14285.638,E2 -14285.638} C_VEL
LIN {X 0,Y 340.74,Z 146.041,A -85,B 0,C 180,E1 -14289.473,E2 -14289.473} C_VEL
LIN {X 0,Y 340.791,Z 146.032,A -85,B 0,C 180,E1 -14291.98,E2 -14291.98} C_VEL
LIN {X 0,Y 340.868,Z 146.023,A -85,B 0,C 180,E1 -14295.705,E2 -14295.705} C_VEL
LIN {X 0,Y 340.87,Z 146.025,A -85,B 0,C 180,E1 -14299.306,E2 -14299.306} C_VEL
LIN {X 0,Y 341.058,Z 146.003,A -85,B 0,C 180,E1 -14302.897,E2 -14302.897} C_VEL
LIN {X 0,Y 341.168,Z 145.985,A -85,B 0,C 180,E1 -14307.638,E2 -14307.638} C_VEL
LIN {X 0,Y 341.295,Z 145.969,A -85,B 0,C 180,E1 -14310,E2 -14310} C_VEL
LIN {X 0,Y 341.168,Z 145.987,A -85,B 0,C 180,E1 -14312.361,E2 -14312.361} C_VEL
LIN {X 0,Y 341.058,Z 146,A -85,B 0,C 180,E1 -14317.102,E2 -14317.102} C_VEL
LIN {X 0,Y 340.869,Z 146.026,A -85,B 0,C 180,E1 -14320.693,E2 -14320.693} C_VEL
LIN {X 0,Y 340.86,Z 146.027,A -85,B 0,C 180,E1 -14324.324,E2 -14324.324} C_VEL
LIN {X 0,Y 340.835,Z 146.031,A -85,B 0,C 180,E1 -14328.467,E2 -14328.467} C_VEL
LIN {X 0,Y 340.7,Z 146.042,A -85,B 0,C 180,E1 -14332.192,E2 -14332.192} C_VEL
LIN {X 0,Y 340.769,Z 146.035,A -85,B 0,C 180,E1 -14335.664,E2 -14335.664} C_VEL
LIN {X 0,Y 340.782,Z 146.032,A -85,B 0,C 180,E1 -14337.332,E2 -14337.332} C_VEL
LIN {X 0,Y 340.08,Z 146.125,A -85,B 0,C 180,E1 -14338.318,E2 -14338.318} C_VEL
LIN {X 0,Y 337.166,Z 146.486,A -85,B 0,C 180,E1 -14339.921,E2 -14339.921} C_VEL
LIN {X 0,Y 334.73,Z 146.787,A -85,B 0,C 180,E1 -14341.219,E2 -14341.219} C_VEL
LIN {X 0,Y 333.714,Z 146.918,A -85,B 0,C 180,E1 -14342.225,E2 -14342.225} C_VEL
LIN {X 0,Y 333.647,Z 146.923,A -85,B 0,C 180,E1 -14342.565,E2 -14342.565} C_VEL
LIN {X 0,Y 333.673,Z 146.923,A -85,B 0,C 180,E1 -14346.139,E2 -14346.139} C_VEL
LIN {X 0,Y 333.678,Z 146.918,A -85,B 0,C 180,E1 -14349.187,E2 -14349.187} C_VEL
LIN {X 0,Y 333.686,Z 146.917,A -85,B 0,C 180,E1 -14352.511,E2 -14352.511} C_VEL
LIN {X 0,Y 333.657,Z 146.925,A -85,B 0,C 180,E1 -14355.966,E2 -14355.966} C_VEL
LIN {X 0,Y 333.653,Z 146.922,A -85,B 0,C 180,E1 -14359.314,E2 -14359.314} C_VEL
LIN {X 0,Y 333.652,Z 146.921,A -85,B 0,C 180,E1 -14362.349,E2 -14362.349} C_VEL
LIN {X 0,Y 333.671,Z 146.921,A -85,B 0,C 180,E1 -14365.341,E2 -14365.341} C_VEL
LIN {X 0,Y 333.694,Z 146.92,A -85,B 0,C 180,E1 -14369.638,E2 -14369.638} C_VEL
LIN {X 0,Y 333.74,Z 146.91,A -85,B 0,C 180,E1 -14372.401,E2 -14372.401} C_VEL
LIN {X 0,Y 333.724,Z 146.915,A -85,B 0,C 180,E1 -14375.091,E2 -14375.091} C_VEL
LIN {X 0,Y 333.679,Z 146.92,A -85,B 0,C 180,E1 -14379.02,E2 -14379.02} C_VEL
LIN {X 0,Y 333.791,Z 146.906,A -85,B 0,C 180,E1 -14381.59,E2 -14381.59} C_VEL
LIN {X 0,Y 333.805,Z 146.904,A -85,B 0,C 180,E1 -14385.577,E2 -14385.577} C_VEL
LIN {X 0,Y 333.831,Z 146.904,A -85,B 0,C 180,E1 -14389.078,E2 -14389.078} C_VEL
LIN {X 0,Y 334.01,Z 146.879,A -85,B 0,C 180,E1 -14392.748,E2 -14392.748} C_VEL
LIN {X 0,Y 333.808,Z 146.905,A -85,B 0,C 180,E1 -14395.17,E2 -14395.17} C_VEL
LIN {X 0,Y 334.105,Z 146.865,A -85,B 0,C 180,E1 -14397.589,E2 -14397.589} C_VEL
LIN {X 0,Y 334.245,Z 146.847,A -85,B 0,C 180,E1 -14400,E2 -14400} C_VEL
LIN {X 0,Y 334.105,Z 146.866,A -85,B 0,C 180,E1 -14402.412,E2 -14402.412} C_VEL
LIN {X 0,Y 334.024,Z 146.876,A -85,B 0,C 180,E1 -14407.253,E2 -14407.253} C_VEL
LIN {X 0,Y 333.832,Z 146.901,A -85,B 0,C 180,E1 -14410.922,E2 -14410.922} C_VEL
LIN {X 0,Y 333.807,Z 146.907,A -85,B 0,C 180,E1 -14414.635,E2 -14414.635} C_VEL
LIN {X 0,Y 333.795,Z 146.907,A -85,B 0,C 180,E1 -14418.656,E2 -14418.656} C_VEL
LIN {X 0,Y 333.655,Z 146.925,A -85,B 0,C 180,E1 -14422.281,E2 -14422.281} C_VEL
LIN {X 0,Y 333.734,Z 146.916,A -85,B 0,C 180,E1 -14426.247,E2 -14426.247} C_VEL
LIN {X 0,Y 333.71,Z 146.914,A -85,B 0,C 180,E1 -14428.973,E2 -14428.973} C_VEL
LIN {X 0,Y 333.645,Z 146.924,A -85,B 0,C 180,E1 -14432.588,E2 -14432.588} C_VEL
LIN {X 0,Y 333.676,Z 146.923,A -85,B 0,C 180,E1 -14436.139,E2 -14436.139} C_VEL
LIN {X 0,Y 333.672,Z 146.918,A -85,B 0,C 180,E1 -14439.189,E2 -14439.189} C_VEL
LIN {X 0,Y 333.666,Z 146.92,A -85,B 0,C 180,E1 -14442.507,E2 -14442.507} C_VEL
LIN {X 0,Y 333.598,Z 146.933,A -85,B 0,C 180,E1 -14445.956,E2 -14445.956} C_VEL
LIN {X 0,Y 333.648,Z 146.923,A -85,B 0,C 180,E1 -14449.316,E2 -14449.316} C_VEL
LIN {X 0,Y 333.666,Z 146.92,A -85,B 0,C 180,E1 -14453.168,E2 -14453.168} C_VEL
LIN {X 0,Y 333.675,Z 146.92,A -85,B 0,C 180,E1 -14455.342,E2 -14455.342} C_VEL
LIN {X 0,Y 333.703,Z 147.024,A -85,B 0,C 180,E1 -14458.572,E2 -14458.572} C_VEL
LIN {X 0,Y 336.509,Z 160.266,A -85,B 0,C 180,E1 -14461.972,E2 -14461.972} C_VEL
LIN {X 0,Y 337.677,Z 167.201,A -85,B 0,C 180,E1 -14463.687,E2 -14463.687} C_VEL
LIN {X 0,Y 336.031,Z 183.514,A -85,B 0,C 180,E1 -14467.408,E2 -14467.408} C_VEL
LIN {X 0,Y 340.76,Z 224.163,A -85,B 0,C 180,E1 -14468.741,E2 -14468.741} C_VEL
LIN {X 0,Y 339.038,Z 293.111,A -85,B 0,C 180,E1 -14470.512,E2 -14470.512} C_VEL
LIN {X 0,Y 338.333,Z 306.705,A -85,B 0,C 180,E1 -14471.1,E2 -14471.1} C_VEL
LIN {X 0,Y 337.473,Z 319.135,A -85,B 0,C 180,E1 -14471.876,E2 -14471.876} C_VEL
LIN {X 0,Y 336.467,Z 330.752,A -85,B 0,C 180,E1 -14472.841,E2 -14472.841} C_VEL
LIN {X 0,Y 335.455,Z 342.105,A -85,B 0,C 180,E1 -14474.04,E2 -14474.04} C_VEL
LIN {X 0,Y 334.469,Z 352.372,A -85,B 0,C 180,E1 -14475.396,E2 -14475.396} C_VEL
LIN {X 0,Y 333.86,Z 359.981,A -85,B 0,C 180,E1 -14476.612,E2 -14476.612} C_VEL
LIN {X 0,Y 333.232,Z 367.929,A -85,B 0,C 180,E1 -14478.134,E2 -14478.134} C_VEL
LIN {X 0,Y 332.601,Z 375.666,A -85,B 0,C 180,E1 -14479.961,E2 -14479.961} C_VEL
LIN {X 0,Y 332.355,Z 380.936,A -85,B 0,C 180,E1 -14481.488,E2 -14481.488} C_VEL
LIN {X 0,Y 332.155,Z 385.996,A -85,B 0,C 180,E1 -14483.318,E2 -14483.318} C_VEL
LIN {X 0,Y 332.158,Z 389.85,A -85,B 0,C 180,E1 -14485.145,E2 -14485.145} C_VEL
LIN {X 0,Y 332.104,Z 391.802,A -85,B 0,C 180,E1 -14486.361,E2 -14486.361} C_VEL
LIN {X 0,Y 332.16,Z 393.299,A -85,B 0,C 180,E1 -14487.575,E2 -14487.575} C_VEL
LIN {X 0,Y 332.269,Z 394.317,A -85,B 0,C 180,E1 -14488.788,E2 -14488.788} C_VEL
LIN {X 0,Y 332.275,Z 394.909,A -85,B 0,C 180,E1 -14490,E2 -14490} C_VEL
LIN {X 0,Y 332.16,Z 395.079,A -85,B 0,C 180,E1 -14491.213,E2 -14491.213} C_VEL
LIN {X 0,Y 332.044,Z 394.798,A -85,B 0,C 180,E1 -14492.427,E2 -14492.427} C_VEL
LIN {X 0,Y 332.041,Z 394.087,A -85,B 0,C 180,E1 -14493.641,E2 -14493.641} C_VEL
LIN {X 0,Y 331.979,Z 391.884,A -85,B 0,C 180,E1 -14495.733,E2 -14495.733} C_VEL
LIN {X 0,Y 332.248,Z 388.24,A -85,B 0,C 180,E1 -14497.903,E2 -14497.903} C_VEL
LIN {X 0,Y 332.666,Z 383.981,A -85,B 0,C 180,E1 -14499.731,E2 -14499.731} C_VEL
LIN {X 0,Y 333.438,Z 377.511,A -85,B 0,C 180,E1 -14501.859,E2 -14501.859} C_VEL
LIN {X 0,Y 334.545,Z 370.518,A -85,B 0,C 180,E1 -14503.671,E2 -14503.671} C_VEL
LIN {X 0,Y 335.755,Z 361.9,A -85,B 0,C 180,E1 -14505.48,E2 -14505.48} C_VEL
LIN {X 0,Y 337.178,Z 353.086,A -85,B 0,C 180,E1 -14506.967,E2 -14506.967} C_VEL
LIN {X 0,Y 338.822,Z 342.318,A -85,B 0,C 180,E1 -14508.441,E2 -14508.441} C_VEL
LIN {X 0,Y 340.502,Z 331.731,A -85,B 0,C 180,E1 -14509.597,E2 -14509.597} C_VEL
LIN {X 0,Y 341.958,Z 320.303,A -85,B 0,C 180,E1 -14510.607,E2 -14510.607} C_VEL
LIN {X 0,Y 343.296,Z 308.797,A -85,B 0,C 180,E1 -14511.387,E2 -14511.387} C_VEL
LIN {X 0,Y 344.644,Z 294.537,A -85,B 0,C 180,E1 -14512.085,E2 -14512.085} C_VEL
LIN {X 0,Y 345.423,Z 278.488,A -85,B 0,C 180,E1 -14512.584,E2 -14512.584} C_VEL
LIN {X 0,Y 347.567,Z 224.22,A -85,B 0,C 180,E1 -14514.039,E2 -14514.039} C_VEL
LIN {X 0,Y 345.514,Z 207.617,A -85,B 0,C 180,E1 -14514.785,E2 -14514.785} C_VEL
LIN {X 0,Y 341.973,Z 188.416,A -85,B 0,C 180,E1 -14515.815,E2 -14515.815} C_VEL
LIN {X 0,Y 339.714,Z 178.524,A -85,B 0,C 180,E1 -14516.451,E2 -14516.451} C_VEL
LIN {X 0,Y 340.242,Z 174.739,A -85,B 0,C 180,E1 -14517.351,E2 -14517.351} C_VEL
LIN {X 0,Y 339.228,Z 168.216,A -85,B 0,C 180,E1 -14519.151,E2 -14519.151} C_VEL
LIN {X 0,Y 336.917,Z 158.302,A -85,B 0,C 180,E1 -14522.135,E2 -14522.135} C_VEL
LIN {X 0,Y 334.14,Z 148.651,A -85,B 0,C 180,E1 -14525.374,E2 -14525.374} C_VEL
LIN {X 0,Y 333.666,Z 146.924,A -85,B 0,C 180,E1 -14526.052,E2 -14526.052} C_VEL
LIN {X 0,Y 333.65,Z 146.927,A -85,B 0,C 180,E1 -14529.192,E2 -14529.192} C_VEL
LIN {X 0,Y 333.636,Z 146.925,A -85,B 0,C 180,E1 -14532.5,E2 -14532.5} C_VEL
LIN {X 0,Y 333.6,Z 146.927,A -85,B 0,C 180,E1 -14535.955,E2 -14535.955} C_VEL
LIN {X 0,Y 333.651,Z 146.919,A -85,B 0,C 180,E1 -14539.315,E2 -14539.315} C_VEL
LIN {X 0,Y 333.668,Z 146.914,A -85,B 0,C 180,E1 -14543.168,E2 -14543.168} C_VEL
LIN {X 0,Y 333.677,Z 146.915,A -85,B 0,C 180,E1 -14545.341,E2 -14545.341} C_VEL
LIN {X 0,Y 333.694,Z 146.917,A -85,B 0,C 180,E1 -14549.637,E2 -14549.637} C_VEL
LIN {X 0,Y 333.743,Z 146.912,A -85,B 0,C 180,E1 -14552.401,E2 -14552.401} C_VEL
LIN {X 0,Y 333.73,Z 146.911,A -85,B 0,C 180,E1 -14555.091,E2 -14555.091} C_VEL
LIN {X 0,Y 333.688,Z 146.916,A -85,B 0,C 180,E1 -14559.019,E2 -14559.019} C_VEL
LIN {X 0,Y 333.745,Z 146.907,A -85,B 0,C 180,E1 -14561.586,E2 -14561.586} C_VEL
LIN {X 0,Y 333.812,Z 146.905,A -85,B 0,C 180,E1 -14565.576,E2 -14565.576} C_VEL
LIN {X 0,Y 333.821,Z 146.902,A -85,B 0,C 180,E1 -14569.077,E2 -14569.077} C_VEL
LIN {X 0,Y 333.971,Z 146.886,A -85,B 0,C 180,E1 -14572.746,E2 -14572.746} C_VEL
LIN {X 0,Y 333.8,Z 146.911,A -85,B 0,C 180,E1 -14575.168,E2 -14575.168} C_VEL
LIN {X 0,Y 333.854,Z 147.092,A -85,B 0,C 180,E1 -14576.228,E2 -14576.228} C_VEL
LIN {X 0,Y 335.591,Z 152.232,A -85,B 0,C 180,E1 -14578.123,E2 -14578.123} C_VEL
LIN {X 0,Y 341.543,Z 162.942,A -85,B 0,C 180,E1 -14579.264,E2 -14579.264} C_VEL
LIN {X 0,Y 346.608,Z 173.84,A -85,B 0,C 180,E1 -14580.22,E2 -14580.22} C_VEL
LIN {X 0,Y 349.205,Z 180.559,A -85,B 0,C 180,E1 -14580.73,E2 -14580.73} C_VEL
LIN {X 0,Y 345.729,Z 259.109,A -85,B 0,C 180,E1 -14582.869,E2 -14582.869} C_VEL
LIN {X 0,Y 344.928,Z 272.542,A -85,B 0,C 180,E1 -14583.476,E2 -14583.476} C_VEL
LIN {X 0,Y 343.958,Z 284.574,A -85,B 0,C 180,E1 -14584.247,E2 -14584.247} C_VEL
LIN {X 0,Y 342.621,Z 296.9,A -85,B 0,C 180,E1 -14585.296,E2 -14585.296} C_VEL
LIN {X 0,Y 341.147,Z 308.077,A -85,B 0,C 180,E1 -14586.505,E2 -14586.505} C_VEL
LIN {X 0,Y 339.825,Z 317.241,A -85,B 0,C 180,E1 -14587.739,E2 -14587.739} C_VEL
LIN {X 0,Y 338.326,Z 326.509,A -85,B 0,C 180,E1 -14589.264,E2 -14589.264} C_VEL
LIN {X 0,Y 337.058,Z 334.181,A -85,B 0,C 180,E1 -14590.816,E2 -14590.816} C_VEL
LIN {X 0,Y 335.687,Z 341.717,A -85,B 0,C 180,E1 -14592.699,E2 -14592.699} C_VEL
LIN {X 0,Y 334.473,Z 348.329,A -85,B 0,C 180,E1 -14594.858,E2 -14594.858} C_VEL
LIN {X 0,Y 333.487,Z 353.522,A -85,B 0,C 180,E1 -14597.159,E2 -14597.159} C_VEL
LIN {X 0,Y 333.032,Z 355.641,A -85,B 0,C 180,E1 -14598.454,E2 -14598.454} C_VEL
LIN {X 0,Y 332.682,Z 357.295,A -85,B 0,C 180,E1 -14599.755,E2 -14599.755} C_VEL
LIN {X 0,Y 332.337,Z 358.702,A -85,B 0,C 180,E1 -14601.49,E2 -14601.49} C_VEL
LIN {X 0,Y 332.07,Z 359.285,A -85,B 0,C 180,E1 -14603.71,E2 -14603.71} C_VEL
LIN {X 0,Y 332.001,Z 358.926,A -85,B 0,C 180,E1 -14605.047,E2 -14605.047} C_VEL
LIN {X 0,Y 331.993,Z 357.273,A -85,B 0,C 180,E1 -14607.239,E2 -14607.239} C_VEL
LIN {X 0,Y 332.231,Z 354.741,A -85,B 0,C 180,E1 -14609.113,E2 -14609.113} C_VEL
LIN {X 0,Y 332.556,Z 350.694,A -85,B 0,C 180,E1 -14611.182,E2 -14611.182} C_VEL
LIN {X 0,Y 332.988,Z 345.031,A -85,B 0,C 180,E1 -14613.281,E2 -14613.281} C_VEL
LIN {X 0,Y 333.52,Z 339.081,A -85,B 0,C 180,E1 -14615.007,E2 -14615.007} C_VEL
LIN {X 0,Y 334.195,Z 331.646,A -85,B 0,C 180,E1 -14616.753,E2 -14616.753} C_VEL
LIN {X 0,Y 334.979,Z 322.837,A -85,B 0,C 180,E1 -14618.429,E2 -14618.429} C_VEL
LIN {X 0,Y 335.934,Z 312.063,A -85,B 0,C 180,E1 -14620.067,E2 -14620.067} C_VEL
LIN {X 0,Y 336.726,Z 302.133,A -85,B 0,C 180,E1 -14621.29,E2 -14621.29} C_VEL
LIN {X 0,Y 337.619,Z 290.088,A -85,B 0,C 180,E1 -14622.471,E2 -14622.471} C_VEL
LIN {X 0,Y 338.429,Z 277.471,A -85,B 0,C 180,E1 -14623.424,E2 -14623.424} C_VEL
LIN {X 0,Y 339.034,Z 264.185,A -85,B 0,C 180,E1 -14624.155,E2 -14624.155} C_VEL
LIN {X 0,Y 339.493,Z 250.357,A -85,B 0,C 180,E1 -14624.65,E2 -14624.65} C_VEL
LIN {X 0,Y 341.472,Z 172.422,A -85,B 0,C 180,E1 -14626.613,E2 -14626.613} C_VEL
LIN {X 0,Y 338.668,Z 162.554,A -85,B 0,C 180,E1 -14627.023,E2 -14627.023} C_VEL
LIN {X 0,Y 333.803,Z 147.507,A -85,B 0,C 180,E1 -14627.694,E2 -14627.694} C_VEL
LIN {X 0,Y 333.722,Z 146.917,A -85,B 0,C 180,E1 -14627.936,E2 -14627.936} C_VEL
LIN {X 0,Y 333.651,Z 146.921,A -85,B 0,C 180,E1 -14632.348,E2 -14632.348} C_VEL
LIN {X 0,Y 333.673,Z 146.922,A -85,B 0,C 180,E1 -14635.341,E2 -14635.341} C_VEL
LIN {X 0,Y 333.702,Z 146.918,A -85,B 0,C 180,E1 -14639.71,E2 -14639.71} C_VEL
LIN {X 0,Y 333.743,Z 146.909,A -85,B 0,C 180,E1 -14642.401,E2 -14642.401} C_VEL
LIN {X 0,Y 333.726,Z 146.915,A -85,B 0,C 180,E1 -14645.09,E2 -14645.09} C_VEL
LIN {X 0,Y 333.676,Z 146.921,A -85,B 0,C 180,E1 -14649.018,E2 -14649.018} C_VEL
LIN {X 0,Y 333.739,Z 146.912,A -85,B 0,C 180,E1 -14651.586,E2 -14651.586} C_VEL
LIN {X 0,Y 333.807,Z 146.903,A -85,B 0,C 180,E1 -14655.576,E2 -14655.576} C_VEL
LIN {X 0,Y 333.833,Z 146.904,A -85,B 0,C 180,E1 -14659.078,E2 -14659.078} C_VEL
LIN {X 0,Y 334.011,Z 146.88,A -85,B 0,C 180,E1 -14662.747,E2 -14662.747} C_VEL
LIN {X 0,Y 333.808,Z 146.905,A -85,B 0,C 180,E1 -14665.169,E2 -14665.169} C_VEL
LIN {X 0,Y 334.106,Z 146.865,A -85,B 0,C 180,E1 -14667.588,E2 -14667.588} C_VEL
LIN {X 0,Y 334.246,Z 146.847,A -85,B 0,C 180,E1 -14670,E2 -14670} C_VEL
LIN {X 0,Y 334.105,Z 146.867,A -85,B 0,C 180,E1 -14672.411,E2 -14672.411} C_VEL
LIN {X 0,Y 334.013,Z 146.876,A -85,B 0,C 180,E1 -14676.039,E2 -14676.039} C_VEL
LIN {X 0,Y 333.982,Z 146.884,A -85,B 0,C 180,E1 -14678.501,E2 -14678.501} C_VEL
LIN {X 0,Y 333.789,Z 146.906,A -85,B 0,C 180,E1 -14682.154,E2 -14682.154} C_VEL
LIN {X 0,Y 333.775,Z 146.906,A -85,B 0,C 180,E1 -14685.886,E2 -14685.886} C_VEL
LIN {X 0,Y 333.794,Z 146.906,A -85,B 0,C 180,E1 -14688.655,E2 -14688.655} C_VEL
LIN {X 0,Y 333.654,Z 146.926,A -85,B 0,C 180,E1 -14692.28,E2 -14692.28} C_VEL
LIN {X 0,Y 333.733,Z 146.917,A -85,B 0,C 180,E1 -14696.246,E2 -14696.246} C_VEL
LIN {X 0,Y 333.709,Z 146.914,A -85,B 0,C 180,E1 -14698.972,E2 -14698.972} C_VEL
LIN {X 0,Y 333.647,Z 146.923,A -85,B 0,C 180,E1 -14702.565,E2 -14702.565} C_VEL
LIN {X 0,Y 333.016,Z 147.004,A -85,B 0,C 180,E1 -14703.572,E2 -14703.572} C_VEL
LIN {X 0,Y 330.162,Z 147.358,A -85,B 0,C 180,E1 -14705.21,E2 -14705.21} C_VEL
LIN {X 0,Y 327.727,Z 147.66,A -85,B 0,C 180,E1 -14706.537,E2 -14706.537} C_VEL
LIN {X 0,Y 326.688,Z 147.79,A -85,B 0,C 180,E1 -14707.564,E2 -14707.564} C_VEL
LIN {X 0,Y 326.609,Z 147.796,A -85,B 0,C 180,E1 -14707.913,E2 -14707.913} C_VEL
LIN {X 0,Y 326.626,Z 147.796,A -85,B 0,C 180,E1 -14711.142,E2 -14711.142} C_VEL
LIN {X 0,Y 326.599,Z 147.799,A -85,B 0,C 180,E1 -14714.756,E2 -14714.756} C_VEL
LIN {X 0,Y 326.599,Z 147.802,A -85,B 0,C 180,E1 -14718.158,E2 -14718.158} C_VEL
LIN {X 0,Y 326.639,Z 147.797,A -85,B 0,C 180,E1 -14721.394,E2 -14721.394} C_VEL
LIN {X 0,Y 326.616,Z 147.797,A -85,B 0,C 180,E1 -14724.851,E2 -14724.851} C_VEL
LIN {X 0,Y 326.607,Z 147.803,A -85,B 0,C 180,E1 -14727.456,E2 -14727.456} C_VEL
LIN {X 0,Y 326.657,Z 147.792,A -85,B 0,C 180,E1 -14730.341,E2 -14730.341} C_VEL
LIN {X 0,Y 326.687,Z 147.788,A -85,B 0,C 180,E1 -14734.517,E2 -14734.517} C_VEL
LIN {X 0,Y 326.644,Z 147.794,A -85,B 0,C 180,E1 -14738.546,E2 -14738.546} C_VEL
LIN {X 0,Y 326.741,Z 147.786,A -85,B 0,C 180,E1 -14741.178,E2 -14741.178} C_VEL
LIN {X 0,Y 326.76,Z 147.783,A -85,B 0,C 180,E1 -14745.433,E2 -14745.433} C_VEL
LIN {X 0,Y 326.767,Z 147.781,A -85,B 0,C 180,E1 -14748.839,E2 -14748.839} C_VEL
LIN {X 0,Y 326.963,Z 147.756,A -85,B 0,C 180,E1 -14752.59,E2 -14752.59} C_VEL
LIN {X 0,Y 326.774,Z 147.782,A -85,B 0,C 180,E1 -14755.065,E2 -14755.065} C_VEL
LIN {X 0,Y 327.045,Z 147.745,A -85,B 0,C 180,E1 -14757.537,E2 -14757.537} C_VEL
LIN {X 0,Y 327.197,Z 147.725,A -85,B 0,C 180,E1 -14760,E2 -14760} C_VEL
LIN {X 0,Y 327.046,Z 147.746,A -85,B 0,C 180,E1 -14762.464,E2 -14762.464} C_VEL
LIN {X 0,Y 326.995,Z 147.751,A -85,B 0,C 180,E1 -14766.17,E2 -14766.17} C_VEL
LIN {X 0,Y 326.913,Z 147.766,A -85,B 0,C 180,E1 -14768.656,E2 -14768.656} C_VEL
LIN {X 0,Y 326.734,Z 147.786,A -85,B 0,C 180,E1 -14772.422,E2 -14772.422} C_VEL
LIN {X 0,Y 326.753,Z 147.782,A -85,B 0,C 180,E1 -14774.958,E2 -14774.958} C_VEL
LIN {X 0,Y 326.731,Z 147.785,A -85,B 0,C 180,E1 -14778.839,E2 -14778.839} C_VEL
LIN {X 0,Y 326.601,Z 147.801,A -85,B 0,C 180,E1 -14782.789,E2 -14782.789} C_VEL
LIN {X 0,Y 326.689,Z 147.788,A -85,B 0,C 180,E1 -14785.484,E2 -14785.484} C_VEL
LIN {X 0,Y 326.66,Z 147.793,A -85,B 0,C 180,E1 -14789.66,E2 -14789.66} C_VEL
LIN {X 0,Y 326.607,Z 147.803,A -85,B 0,C 180,E1 -14794.02,E2 -14794.02} C_VEL
LIN {X 0,Y 326.629,Z 147.796,A -85,B 0,C 180,E1 -14797.24,E2 -14797.24} C_VEL
LIN {X 0,Y 326.604,Z 147.802,A -85,B 0,C 180,E1 -14800.208,E2 -14800.208} C_VEL
LIN {X 0,Y 326.578,Z 147.804,A -85,B 0,C 180,E1 -14803.523,E2 -14803.523} C_VEL
LIN {X 0,Y 326.576,Z 147.802,A -85,B 0,C 180,E1 -14807.029,E2 -14807.029} C_VEL
LIN {X 0,Y 326.612,Z 147.798,A -85,B 0,C 180,E1 -14810.773,E2 -14810.773} C_VEL
LIN {X 0,Y 326.613,Z 147.798,A -85,B 0,C 180,E1 -14814.481,E2 -14814.481} C_VEL
LIN {X 0,Y 326.656,Z 147.816,A -85,B 0,C 180,E1 -14818.28,E2 -14818.28} C_VEL
LIN {X 0,Y 329.652,Z 162.14,A -85,B 0,C 180,E1 -14822.029,E2 -14822.029} C_VEL
LIN {X 0,Y 330.646,Z 167.915,A -85,B 0,C 180,E1 -14823.49,E2 -14823.49} C_VEL
LIN {X 0,Y 329.103,Z 183.027,A -85,B 0,C 180,E1 -14827.038,E2 -14827.038} C_VEL
LIN {X 0,Y 333.934,Z 224.35,A -85,B 0,C 180,E1 -14828.425,E2 -14828.425} C_VEL
LIN {X 0,Y 332.168,Z 292.102,A -85,B 0,C 180,E1 -14830.213,E2 -14830.213} C_VEL
LIN {X 0,Y 331.419,Z 305.825,A -85,B 0,C 180,E1 -14830.811,E2 -14830.811} C_VEL
LIN {X 0,Y 330.567,Z 317.871,A -85,B 0,C 180,E1 -14831.564,E2 -14831.564} C_VEL
LIN {X 0,Y 329.607,Z 328.88,A -85,B 0,C 180,E1 -14832.472,E2 -14832.472} C_VEL
LIN {X 0,Y 328.557,Z 340.488,A -85,B 0,C 180,E1 -14833.695,E2 -14833.695} C_VEL
LIN {X 0,Y 327.516,Z 351.005,A -85,B 0,C 180,E1 -14835.079,E2 -14835.079} C_VEL
LIN {X 0,Y 326.724,Z 360.488,A -85,B 0,C 180,E1 -14836.631,E2 -14836.631} C_VEL
LIN {X 0,Y 326.088,Z 368.28,A -85,B 0,C 180,E1 -14838.186,E2 -14838.186} C_VEL
LIN {X 0,Y 325.489,Z 375.889,A -85,B 0,C 180,E1 -14840.053,E2 -14840.053} C_VEL
LIN {X 0,Y 325.205,Z 381.977,A -85,B 0,C 180,E1 -14841.925,E2 -14841.925} C_VEL
LIN {X 0,Y 325.098,Z 387.069,A -85,B 0,C 180,E1 -14843.955,E2 -14843.955} C_VEL
LIN {X 0,Y 325.07,Z 389.202,A -85,B 0,C 180,E1 -14845.039,E2 -14845.039} C_VEL
LIN {X 0,Y 325.031,Z 391.197,A -85,B 0,C 180,E1 -14846.281,E2 -14846.281} C_VEL
LIN {X 0,Y 325.068,Z 392.752,A -85,B 0,C 180,E1 -14847.522,E2 -14847.522} C_VEL
LIN {X 0,Y 325.19,Z 393.826,A -85,B 0,C 180,E1 -14848.762,E2 -14848.762} C_VEL
LIN {X 0,Y 325.214,Z 394.455,A -85,B 0,C 180,E1 -14850,E2 -14850} C_VEL
LIN {X 0,Y 325.066,Z 394.657,A -85,B 0,C 180,E1 -14851.239,E2 -14851.239} C_VEL
LIN {X 0,Y 324.956,Z 394.439,A -85,B 0,C 180,E1 -14852.48,E2 -14852.48} C_VEL
LIN {X 0,Y 324.963,Z 393.765,A -85,B 0,C 180,E1 -14853.72,E2 -14853.72} C_VEL
LIN {X 0,Y 324.879,Z 391.871,A -85,B 0,C 180,E1 -14855.668,E2 -14855.668} C_VEL
LIN {X 0,Y 325.185,Z 388.057,A -85,B 0,C 180,E1 -14858.076,E2 -14858.076} C_VEL
LIN {X 0,Y 325.62,Z 383.891,A -85,B 0,C 180,E1 -14859.943,E2 -14859.943} C_VEL
LIN {X 0,Y 326.481,Z 377.554,A -85,B 0,C 180,E1 -14862.116,E2 -14862.116} C_VEL
LIN {X 0,Y 327.647,Z 370.65,A -85,B 0,C 180,E1 -14863.964,E2 -14863.964} C_VEL
LIN {X 0,Y 329.011,Z 361.621,A -85,B 0,C 180,E1 -14865.911,E2 -14865.911} C_VEL
LIN {X 0,Y 330.728,Z 351.553,A -85,B 0,C 180,E1 -14867.627,E2 -14867.627} C_VEL
LIN {X 0,Y 332.592,Z 340.635,A -85,B 0,C 180,E1 -14869.119,E2 -14869.119} C_VEL
LIN {X 0,Y 334.356,Z 329.807,A -85,B 0,C 180,E1 -14870.293,E2 -14870.293} C_VEL
LIN {X 0,Y 335.845,Z 317.958,A -85,B 0,C 180,E1 -14871.322,E2 -14871.322} C_VEL
LIN {X 0,Y 337.497,Z 304.675,A -85,B 0,C 180,E1 -14872.175,E2 -14872.175} C_VEL
LIN {X 0,Y 338.73,Z 290.299,A -85,B 0,C 180,E1 -14872.814,E2 -14872.814} C_VEL
LIN {X 0,Y 341.521,Z 224.833,A -85,B 0,C 180,E1 -14874.655,E2 -14874.655} C_VEL
LIN {X 0,Y 339.424,Z 207.858,A -85,B 0,C 180,E1 -14875.458,E2 -14875.458} C_VEL
LIN {X 0,Y 335.655,Z 187.93,A -85,B 0,C 180,E1 -14876.589,E2 -14876.589} C_VEL
LIN {X 0,Y 333.343,Z 178.018,A -85,B 0,C 180,E1 -14877.261,E2 -14877.261} C_VEL
LIN {X 0,Y 333.481,Z 175.284,A -85,B 0,C 180,E1 -14877.963,E2 -14877.963} C_VEL
LIN {X 0,Y 331.685,Z 166.466,A -85,B 0,C 180,E1 -14880.566,E2 -14880.566} C_VEL
LIN {X 0,Y 329.623,Z 157.979,A -85,B 0,C 180,E1 -14883.284,E2 -14883.284} C_VEL
LIN {X 0,Y 327.195,Z 149.807,A -85,B 0,C 180,E1 -14886.206,E2 -14886.206} C_VEL
LIN {X 0,Y 326.634,Z 147.799,A -85,B 0,C 180,E1 -14887.047,E2 -14887.047} C_VEL
LIN {X 0,Y 326.595,Z 147.802,A -85,B 0,C 180,E1 -14890.209,E2 -14890.209} C_VEL
LIN {X 0,Y 326.565,Z 147.806,A -85,B 0,C 180,E1 -14893.525,E2 -14893.525} C_VEL
LIN {X 0,Y 326.58,Z 147.803,A -85,B 0,C 180,E1 -14897.028,E2 -14897.028} C_VEL
LIN {X 0,Y 326.615,Z 147.792,A -85,B 0,C 180,E1 -14900.773,E2 -14900.773} C_VEL
LIN {X 0,Y 326.616,Z 147.796,A -85,B 0,C 180,E1 -14904.48,E2 -14904.48} C_VEL
LIN {X 0,Y 326.611,Z 147.8,A -85,B 0,C 180,E1 -14907.455,E2 -14907.455} C_VEL
LIN {X 0,Y 326.651,Z 147.795,A -85,B 0,C 180,E1 -14910.34,E2 -14910.34} C_VEL
LIN {X 0,Y 326.693,Z 147.784,A -85,B 0,C 180,E1 -14914.516,E2 -14914.516} C_VEL
LIN {X 0,Y 326.651,Z 147.796,A -85,B 0,C 180,E1 -14918.545,E2 -14918.545} C_VEL
LIN {X 0,Y 326.71,Z 147.787,A -85,B 0,C 180,E1 -14921.175,E2 -14921.175} C_VEL
LIN {X 0,Y 326.766,Z 147.783,A -85,B 0,C 180,E1 -14925.433,E2 -14925.433} C_VEL
LIN {X 0,Y 326.762,Z 147.78,A -85,B 0,C 180,E1 -14928.838,E2 -14928.838} C_VEL
LIN {X 0,Y 326.926,Z 147.763,A -85,B 0,C 180,E1 -14932.589,E2 -14932.589} C_VEL
LIN {X 0,Y 326.783,Z 147.902,A -85,B 0,C 180,E1 -14935.219,E2 -14935.219} C_VEL
LIN {X 0,Y 328.431,Z 152.753,A -85,B 0,C 180,E1 -14937.144,E2 -14937.144} C_VEL
LIN {X 0,Y 335.78,Z 165.644,A -85,B 0,C 180,E1 -14938.631,E2 -14938.631} C_VEL
LIN {X 0,Y 341.049,Z 176.85,A -85,B 0,C 180,E1 -14939.679,E2 -14939.679} C_VEL
LIN {X 0,Y 343.212,Z 182.565,A -85,B 0,C 180,E1 -14940.122,E2 -14940.122} C_VEL
LIN {X 0,Y 339.554,Z 259.915,A -85,B 0,C 180,E1 -14942.298,E2 -14942.298} C_VEL
LIN {X 0,Y 338.814,Z 272.193,A -85,B 0,C 180,E1 -14942.864,E2 -14942.864} C_VEL
LIN {X 0,Y 337.764,Z 284.544,A -85,B 0,C 180,E1 -14943.653,E2 -14943.653} C_VEL
LIN {X 0,Y 336.371,Z 296.822,A -85,B 0,C 180,E1 -14944.702,E2 -14944.702} C_VEL
LIN {X 0,Y 334.71,Z 308.882,A -85,B 0,C 180,E1 -14946.026,E2 -14946.026} C_VEL
LIN {X 0,Y 333.024,Z 319.667,A -85,B 0,C 180,E1 -14947.548,E2 -14947.548} C_VEL
LIN {X 0,Y 331.414,Z 328.824,A -85,B 0,C 180,E1 -14949.151,E2 -14949.151} C_VEL
LIN {X 0,Y 330.086,Z 336.164,A -85,B 0,C 180,E1 -14950.736,E2 -14950.736} C_VEL
LIN {X 0,Y 328.667,Z 343.354,A -85,B 0,C 180,E1 -14952.66,E2 -14952.66} C_VEL
LIN {X 0,Y 327.398,Z 349.862,A -85,B 0,C 180,E1 -14954.927,E2 -14954.927} C_VEL
LIN {X 0,Y 326.533,Z 354.032,A -85,B 0,C 180,E1 -14956.891,E2 -14956.891} C_VEL
LIN {X 0,Y 325.847,Z 357.019,A -85,B 0,C 180,E1 -14958.876,E2 -14958.876} C_VEL
LIN {X 0,Y 325.491,Z 358.378,A -85,B 0,C 180,E1 -14960.21,E2 -14960.21} C_VEL
LIN {X 0,Y 325.248,Z 359.349,A -85,B 0,C 180,E1 -14961.696,E2 -14961.696} C_VEL
LIN {X 0,Y 325.076,Z 359.663,A -85,B 0,C 180,E1 -14962.901,E2 -14962.901} C_VEL
LIN {X 0,Y 324.949,Z 359.43,A -85,B 0,C 180,E1 -14964.717,E2 -14964.717} C_VEL
LIN {X 0,Y 324.893,Z 357.815,A -85,B 0,C 180,E1 -14967.017,E2 -14967.017} C_VEL
LIN {X 0,Y 325.139,Z 355.087,A -85,B 0,C 180,E1 -14969.1,E2 -14969.1} C_VEL
LIN {X 0,Y 325.489,Z 351.011,A -85,B 0,C 180,E1 -14971.212,E2 -14971.212} C_VEL
LIN {X 0,Y 325.93,Z 345.311,A -85,B 0,C 180,E1 -14973.356,E2 -14973.356} C_VEL
LIN {X 0,Y 326.475,Z 339.352,A -85,B 0,C 180,E1 -14975.112,E2 -14975.112} C_VEL
LIN {X 0,Y 327.183,Z 331.523,A -85,B 0,C 180,E1 -14976.973,E2 -14976.973} C_VEL
LIN {X 0,Y 327.985,Z 322.962,A -85,B 0,C 180,E1 -14978.614,E2 -14978.614} C_VEL
LIN {X 0,Y 328.938,Z 312.296,A -85,B 0,C 180,E1 -14980.264,E2 -14980.264} C_VEL
LIN {X 0,Y 329.823,Z 301.664,A -85,B 0,C 180,E1 -14981.587,E2 -14981.587} C_VEL
LIN {X 0,Y 330.646,Z 290.641,A -85,B 0,C 180,E1 -14982.682,E2 -14982.682} C_VEL
LIN {X 0,Y 331.505,Z 277.513,A -85,B 0,C 180,E1 -14983.692,E2 -14983.692} C_VEL
LIN {X 0,Y 332.126,Z 264.396,A -85,B 0,C 180,E1 -14984.423,E2 -14984.423} C_VEL
LIN {X 0,Y 332.592,Z 250.503,A -85,B 0,C 180,E1 -14984.929,E2 -14984.929} C_VEL
LIN {X 0,Y 334.662,Z 173.332,A -85,B 0,C 180,E1 -14986.928,E2 -14986.928} C_VEL
LIN {X 0,Y 328.016,Z 152.09,A -85,B 0,C 180,E1 -14987.863,E2 -14987.863} C_VEL
LIN {X 0,Y 326.68,Z 147.793,A -85,B 0,C 180,E1 -14988.092,E2 -14988.092} C_VEL
LIN {X 0,Y 326.623,Z 147.8,A -85,B 0,C 180,E1 -14991.391,E2 -14991.391} C_VEL
LIN {X 0,Y 326.618,Z 147.797,A -85,B 0,C 180,E1 -14994.851,E2 -14994.851} C_VEL
LIN {X 0,Y 326.607,Z 147.804,A -85,B 0,C 180,E1 -14997.455,E2 -14997.455} C_VEL
LIN {X 0,Y 326.66,Z 147.792,A -85,B 0,C 180,E1 -15000.34,E2 -15000.34} C_VEL
LIN {X 0,Y 326.689,Z 147.788,A -85,B 0,C 180,E1 -15004.516,E2 -15004.516} C_VEL
LIN {X 0,Y 326.643,Z 147.794,A -85,B 0,C 180,E1 -15008.545,E2 -15008.545} C_VEL
LIN {X 0,Y 326.706,Z 147.791,A -85,B 0,C 180,E1 -15011.175,E2 -15011.175} C_VEL
LIN {X 0,Y 326.762,Z 147.782,A -85,B 0,C 180,E1 -15015.433,E2 -15015.433} C_VEL
LIN {X 0,Y 326.769,Z 147.782,A -85,B 0,C 180,E1 -15018.838,E2 -15018.838} C_VEL
LIN {X 0,Y 326.965,Z 147.756,A -85,B 0,C 180,E1 -15022.59,E2 -15022.59} C_VEL
LIN {X 0,Y 326.775,Z 147.782,A -85,B 0,C 180,E1 -15025.064,E2 -15025.064} C_VEL
LIN {X 0,Y 327.046,Z 147.744,A -85,B 0,C 180,E1 -15027.536,E2 -15027.536} C_VEL
LIN {X 0,Y 327.197,Z 147.725,A -85,B 0,C 180,E1 -15030,E2 -15030} C_VEL
LIN {X 0,Y 327.045,Z 147.747,A -85,B 0,C 180,E1 -15032.463,E2 -15032.463} C_VEL
LIN {X 0,Y 326.988,Z 147.752,A -85,B 0,C 180,E1 -15036.169,E2 -15036.169} C_VEL
LIN {X 0,Y 326.912,Z 147.766,A -85,B 0,C 180,E1 -15038.655,E2 -15038.655} C_VEL
LIN {X 0,Y 326.733,Z 147.787,A -85,B 0,C 180,E1 -15042.421,E2 -15042.421} C_VEL
LIN {X 0,Y 326.752,Z 147.782,A -85,B 0,C 180,E1 -15044.957,E2 -15044.957} C_VEL
LIN {X 0,Y 326.73,Z 147.785,A -85,B 0,C 180,E1 -15048.838,E2 -15048.838} C_VEL
LIN {X 0,Y 326.6,Z 147.801,A -85,B 0,C 180,E1 -15052.788,E2 -15052.788} C_VEL
LIN {X 0,Y 326.687,Z 147.789,A -85,B 0,C 180,E1 -15055.483,E2 -15055.483} C_VEL
LIN {X 0,Y 326.67,Z 147.796,A -85,B 0,C 180,E1 -15058.249,E2 -15058.249} C_VEL
LIN {X 0,Y 326.598,Z 147.799,A -85,B 0,C 180,E1 -15061.094,E2 -15061.094} C_VEL
LIN {X 0,Y 326.606,Z 147.804,A -85,B 0,C 180,E1 -15064.019,E2 -15064.019} C_VEL
LIN {X 0,Y 326.609,Z 147.796,A -85,B 0,C 180,E1 -15067.913,E2 -15067.913} C_VEL
LIN {X 0,Y 325.957,Z 147.88,A -85,B 0,C 180,E1 -15068.943,E2 -15068.943} C_VEL
LIN {X 0,Y 323.114,Z 148.234,A -85,B 0,C 180,E1 -15070.619,E2 -15070.619} C_VEL
LIN {X 0,Y 320.702,Z 148.539,A -85,B 0,C 180,E1 -15071.977,E2 -15071.977} C_VEL
LIN {X 0,Y 319.676,Z 148.662,A -85,B 0,C 180,E1 -15073.029,E2 -15073.029} C_VEL
LIN {X 0,Y 319.598,Z 148.673,A -85,B 0,C 180,E1 -15073.385,E2 -15073.385} C_VEL
LIN {X 0,Y 319.59,Z 148.673,A -85,B 0,C 180,E1 -15077.023,E2 -15077.023} C_VEL
LIN {X 0,Y 319.578,Z 148.675,A -85,B 0,C 180,E1 -15080.376,E2 -15080.376} C_VEL
LIN {X 0,Y 319.556,Z 148.681,A -85,B 0,C 180,E1 -15083.573,E2 -15083.573} C_VEL
LIN {X 0,Y 319.574,Z 148.674,A -85,B 0,C 180,E1 -15086.686,E2 -15086.686} C_VEL
LIN {X 0,Y 319.588,Z 148.677,A -85,B 0,C 180,E1 -15089.617,E2 -15089.617} C_VEL
LIN {X 0,Y 319.605,Z 148.67,A -85,B 0,C 180,E1 -15092.498,E2 -15092.498} C_VEL
LIN {X 0,Y 319.602,Z 148.676,A -85,B 0,C 180,E1 -15095.304,E2 -15095.304} C_VEL
LIN {X 0,Y 319.594,Z 148.672,A -85,B 0,C 180,E1 -15098.048,E2 -15098.048} C_VEL
LIN {X 0,Y 319.686,Z 148.663,A -85,B 0,C 180,E1 -15100.962,E2 -15100.962} C_VEL
LIN {X 0,Y 319.728,Z 148.66,A -85,B 0,C 180,E1 -15105.276,E2 -15105.276} C_VEL
LIN {X 0,Y 319.754,Z 148.652,A -85,B 0,C 180,E1 -15109.873,E2 -15109.873} C_VEL
LIN {X 0,Y 319.922,Z 148.632,A -85,B 0,C 180,E1 -15112.426,E2 -15112.426} C_VEL
LIN {X 0,Y 319.744,Z 148.659,A -85,B 0,C 180,E1 -15114.956,E2 -15114.956} C_VEL
LIN {X 0,Y 319.989,Z 148.624,A -85,B 0,C 180,E1 -15117.483,E2 -15117.483} C_VEL
LIN {X 0,Y 320.149,Z 148.603,A -85,B 0,C 180,E1 -15120,E2 -15120} C_VEL
LIN {X 0,Y 319.989,Z 148.625,A -85,B 0,C 180,E1 -15122.518,E2 -15122.518} C_VEL
LIN {X 0,Y 319.95,Z 148.629,A -85,B 0,C 180,E1 -15126.306,E2 -15126.306} C_VEL
LIN {X 0,Y 319.841,Z 148.645,A -85,B 0,C 180,E1 -15128.848,E2 -15128.848} C_VEL
LIN {X 0,Y 319.681,Z 148.666,A -85,B 0,C 180,E1 -15132.7,E2 -15132.7} C_VEL
LIN {X 0,Y 319.698,Z 148.659,A -85,B 0,C 180,E1 -15135.296,E2 -15135.296} C_VEL
LIN {X 0,Y 319.672,Z 148.662,A -85,B 0,C 180,E1 -15139.256,E2 -15139.256} C_VEL
LIN {X 0,Y 319.559,Z 148.676,A -85,B 0,C 180,E1 -15143.321,E2 -15143.321} C_VEL
LIN {X 0,Y 319.634,Z 148.67,A -85,B 0,C 180,E1 -15146.089,E2 -15146.089} C_VEL
LIN {X 0,Y 319.588,Z 148.673,A -85,B 0,C 180,E1 -15148.934,E2 -15148.934} C_VEL
LIN {X 0,Y 319.532,Z 148.682,A -85,B 0,C 180,E1 -15151.862,E2 -15151.862} C_VEL
LIN {X 0,Y 319.579,Z 148.675,A -85,B 0,C 180,E1 -15155.544,E2 -15155.544} C_VEL
LIN {X 0,Y 319.597,Z 148.677,A -85,B 0,C 180,E1 -15158.005,E2 -15158.005} C_VEL
LIN {X 0,Y 319.569,Z 148.677,A -85,B 0,C 180,E1 -15161.606,E2 -15161.606} C_VEL
LIN {X 0,Y 319.492,Z 148.685,A -85,B 0,C 180,E1 -15165.259,E2 -15165.259} C_VEL
LIN {X 0,Y 319.528,Z 148.68,A -85,B 0,C 180,E1 -15168.712,E2 -15168.712} C_VEL
LIN {X 0,Y 319.562,Z 148.677,A -85,B 0,C 180,E1 -15172.349,E2 -15172.349} C_VEL
LIN {X 0,Y 319.561,Z 148.677,A -85,B 0,C 180,E1 -15175.124,E2 -15175.124} C_VEL
LIN {X 0,Y 319.622,Z 148.72,A -85,B 0,C 180,E1 -15178.01,E2 -15178.01} C_VEL
LIN {X 0,Y 322.514,Z 162.527,A -85,B 0,C 180,E1 -15181.709,E2 -15181.709} C_VEL
LIN {X 0,Y 323.541,Z 168.092,A -85,B 0,C 180,E1 -15183.152,E2 -15183.152} C_VEL
LIN {X 0,Y 323.314,Z 172.522,A -85,B 0,C 180,E1 -15184.231,E2 -15184.231} C_VEL
LIN {X 0,Y 322.176,Z 182.682,A -85,B 0,C 180,E1 -15186.664,E2 -15186.664} C_VEL
LIN {X 0,Y 327.045,Z 224.269,A -85,B 0,C 180,E1 -15188.108,E2 -15188.108} C_VEL
LIN {X 0,Y 325.255,Z 291.843,A -85,B 0,C 180,E1 -15189.939,E2 -15189.939} C_VEL
LIN {X 0,Y 324.493,Z 305.506,A -85,B 0,C 180,E1 -15190.55,E2 -15190.55} C_VEL
LIN {X 0,Y 323.621,Z 317.526,A -85,B 0,C 180,E1 -15191.318,E2 -15191.318} C_VEL
LIN {X 0,Y 322.639,Z 328.524,A -85,B 0,C 180,E1 -15192.245,E2 -15192.245} C_VEL
LIN {X 0,Y 321.557,Z 340.126,A -85,B 0,C 180,E1 -15193.494,E2 -15193.494} C_VEL
LIN {X 0,Y 320.454,Z 350.944,A -85,B 0,C 180,E1 -15194.951,E2 -15194.951} C_VEL
LIN {X 0,Y 319.772,Z 359.284,A -85,B 0,C 180,E1 -15196.334,E2 -15196.334} C_VEL
LIN {X 0,Y 319.105,Z 367.222,A -85,B 0,C 180,E1 -15197.923,E2 -15197.923} C_VEL
LIN {X 0,Y 318.456,Z 374.951,A -85,B 0,C 180,E1 -15199.832,E2 -15199.832} C_VEL
LIN {X 0,Y 318.153,Z 381.146,A -85,B 0,C 180,E1 -15201.745,E2 -15201.745} C_VEL
LIN {X 0,Y 318.029,Z 386.655,A -85,B 0,C 180,E1 -15203.958,E2 -15203.958} C_VEL
LIN {X 0,Y 317.958,Z 390.592,A -85,B 0,C 180,E1 -15206.198,E2 -15206.198} C_VEL
LIN {X 0,Y 317.978,Z 392.186,A -85,B 0,C 180,E1 -15207.467,E2 -15207.467} C_VEL
LIN {X 0,Y 318.097,Z 393.333,A -85,B 0,C 180,E1 -15208.734,E2 -15208.734} C_VEL
LIN {X 0,Y 318.154,Z 394,A -85,B 0,C 180,E1 -15210,E2 -15210} C_VEL
LIN {X 0,Y 317.972,Z 394.235,A -85,B 0,C 180,E1 -15211.267,E2 -15211.267} C_VEL
LIN {X 0,Y 317.87,Z 394.06,A -85,B 0,C 180,E1 -15212.535,E2 -15212.535} C_VEL
LIN {X 0,Y 317.863,Z 393.447,A -85,B 0,C 180,E1 -15213.804,E2 -15213.804} C_VEL
LIN {X 0,Y 317.804,Z 391.811,A -85,B 0,C 180,E1 -15215.645,E2 -15215.645} C_VEL
LIN {X 0,Y 318.143,Z 387.899,A -85,B 0,C 180,E1 -15218.256,E2 -15218.256} C_VEL
LIN {X 0,Y 318.585,Z 383.81,A -85,B 0,C 180,E1 -15220.165,E2 -15220.165} C_VEL
LIN {X 0,Y 319.506,Z 377.596,A -85,B 0,C 180,E1 -15222.385,E2 -15222.385} C_VEL
LIN {X 0,Y 320.761,Z 370.803,A -85,B 0,C 180,E1 -15224.27,E2 -15224.27} C_VEL
LIN {X 0,Y 322.179,Z 362.062,A -85,B 0,C 180,E1 -15226.234,E2 -15226.234} C_VEL
LIN {X 0,Y 324.009,Z 352.125,A -85,B 0,C 180,E1 -15228.005,E2 -15228.005} C_VEL
LIN {X 0,Y 325.931,Z 341.389,A -85,B 0,C 180,E1 -15229.526,E2 -15229.526} C_VEL
LIN {X 0,Y 327.759,Z 330.854,A -85,B 0,C 180,E1 -15230.72,E2 -15230.72} C_VEL
LIN {X 0,Y 329.315,Z 319.446,A -85,B 0,C 180,E1 -15231.766,E2 -15231.766} C_VEL
LIN {X 0,Y 331.024,Z 306.8,A -85,B 0,C 180,E1 -15232.633,E2 -15232.633} C_VEL
LIN {X 0,Y 332.349,Z 293.19,A -85,B 0,C 180,E1 -15233.318,E2 -15233.318} C_VEL
LIN {X 0,Y 333.355,Z 275.641,A -85,B 0,C 180,E1 -15233.872,E2 -15233.872} C_VEL
LIN {X 0,Y 335.568,Z 225.789,A -85,B 0,C 180,E1 -15235.288,E2 -15235.288} C_VEL
LIN {X 0,Y 333.435,Z 208.497,A -85,B 0,C 180,E1 -15236.137,E2 -15236.137} C_VEL
LIN {X 0,Y 329.807,Z 189.264,A -85,B 0,C 180,E1 -15237.296,E2 -15237.296} C_VEL
LIN {X 0,Y 326.912,Z 177.845,A -85,B 0,C 180,E1 -15238.119,E2 -15238.119} C_VEL
LIN {X 0,Y 325.845,Z 172.189,A -85,B 0,C 180,E1 -15239.741,E2 -15239.741} C_VEL
LIN {X 0,Y 323.589,Z 162.431,A -85,B 0,C 180,E1 -15242.887,E2 -15242.887} C_VEL
LIN {X 0,Y 320.975,Z 153.201,A -85,B 0,C 180,E1 -15246.242,E2 -15246.242} C_VEL
LIN {X 0,Y 319.566,Z 148.68,A -85,B 0,C 180,E1 -15248.11,E2 -15248.11} C_VEL
LIN {X 0,Y 319.529,Z 148.683,A -85,B 0,C 180,E1 -15251.597,E2 -15251.597} C_VEL
LIN {X 0,Y 319.491,Z 148.689,A -85,B 0,C 180,E1 -15255.257,E2 -15255.257} C_VEL
LIN {X 0,Y 319.531,Z 148.675,A -85,B 0,C 180,E1 -15258.712,E2 -15258.712} C_VEL
LIN {X 0,Y 319.58,Z 148.672,A -85,B 0,C 180,E1 -15262.344,E2 -15262.344} C_VEL
LIN {X 0,Y 319.564,Z 148.675,A -85,B 0,C 180,E1 -15265.123,E2 -15265.123} C_VEL
LIN {X 0,Y 319.569,Z 148.671,A -85,B 0,C 180,E1 -15269.059,E2 -15269.059} C_VEL
LIN {X 0,Y 319.609,Z 148.673,A -85,B 0,C 180,E1 -15272.498,E2 -15272.498} C_VEL
LIN {X 0,Y 319.609,Z 148.673,A -85,B 0,C 180,E1 -15275.304,E2 -15275.304} C_VEL
LIN {X 0,Y 319.601,Z 148.674,A -85,B 0,C 180,E1 -15278.048,E2 -15278.048} C_VEL
LIN {X 0,Y 319.661,Z 148.667,A -85,B 0,C 180,E1 -15280.978,E2 -15280.978} C_VEL
LIN {X 0,Y 319.715,Z 148.66,A -85,B 0,C 180,E1 -15285.289,E2 -15285.289} C_VEL
LIN {X 0,Y 319.718,Z 148.658,A -85,B 0,C 180,E1 -15288.589,E2 -15288.589} C_VEL
LIN {X 0,Y 319.882,Z 148.641,A -85,B 0,C 180,E1 -15292.425,E2 -15292.425} C_VEL
LIN {X 0,Y 319.877,Z 148.815,A -85,B 0,C 180,E1 -15294.167,E2 -15294.167} C_VEL
LIN {X 0,Y 321.226,Z 153.572,A -85,B 0,C 180,E1 -15296.079,E2 -15296.079} C_VEL
LIN {X 0,Y 326.574,Z 162.107,A -85,B 0,C 180,E1 -15297.236,E2 -15297.236} C_VEL
LIN {X 0,Y 331.436,Z 170.979,A -85,B 0,C 180,E1 -15298.252,E2 -15298.252} C_VEL
LIN {X 0,Y 336.378,Z 182.023,A -85,B 0,C 180,E1 -15299.294,E2 -15299.294} C_VEL
LIN {X 0,Y 337.244,Z 184.328,A -85,B 0,C 180,E1 -15299.485,E2 -15299.485} C_VEL
LIN {X 0,Y 333.536,Z 260.045,A -85,B 0,C 180,E1 -15301.66,E2 -15301.66} C_VEL
LIN {X 0,Y 332.705,Z 272.953,A -85,B 0,C 180,E1 -15302.269,E2 -15302.269} C_VEL
LIN {X 0,Y 331.501,Z 285.744,A -85,B 0,C 180,E1 -15303.116,E2 -15303.116} C_VEL
LIN {X 0,Y 330.114,Z 297.157,A -85,B 0,C 180,E1 -15304.12,E2 -15304.12} C_VEL
LIN {X 0,Y 328.469,Z 308.427,A -85,B 0,C 180,E1 -15305.371,E2 -15305.371} C_VEL
LIN {X 0,Y 326.832,Z 318.447,A -85,B 0,C 180,E1 -15306.759,E2 -15306.759} C_VEL
LIN {X 0,Y 325.153,Z 327.711,A -85,B 0,C 180,E1 -15308.357,E2 -15308.357} C_VEL
LIN {X 0,Y 323.67,Z 335.459,A -85,B 0,C 180,E1 -15310.003,E2 -15310.003} C_VEL
LIN {X 0,Y 322.158,Z 342.677,A -85,B 0,C 180,E1 -15311.897,E2 -15311.897} C_VEL
LIN {X 0,Y 320.839,Z 348.743,A -85,B 0,C 180,E1 -15313.942,E2 -15313.942} C_VEL
LIN {X 0,Y 319.84,Z 353.281,A -85,B 0,C 180,E1 -15315.942,E2 -15315.942} C_VEL
LIN {X 0,Y 319.062,Z 356.627,A -85,B 0,C 180,E1 -15317.961,E2 -15317.961} C_VEL
LIN {X 0,Y 318.65,Z 358.247,A -85,B 0,C 180,E1 -15319.319,E2 -15319.319} C_VEL
LIN {X 0,Y 318.311,Z 359.345,A -85,B 0,C 180,E1 -15320.687,E2 -15320.687} C_VEL
LIN {X 0,Y 318.111,Z 359.958,A -85,B 0,C 180,E1 -15322.06,E2 -15322.06} C_VEL
LIN {X 0,Y 317.936,Z 360.111,A -85,B 0,C 180,E1 -15323.446,E2 -15323.446} C_VEL
LIN {X 0,Y 317.847,Z 359.655,A -85,B 0,C 180,E1 -15324.965,E2 -15324.965} C_VEL
LIN {X 0,Y 317.794,Z 358.838,A -85,B 0,C 180,E1 -15326.25,E2 -15326.25} C_VEL
LIN {X 0,Y 317.889,Z 357.2,A -85,B 0,C 180,E1 -15327.829,E2 -15327.829} C_VEL
LIN {X 0,Y 318.163,Z 354.208,A -85,B 0,C 180,E1 -15329.802,E2 -15329.802} C_VEL
LIN {X 0,Y 318.534,Z 349.592,A -85,B 0,C 180,E1 -15331.973,E2 -15331.973} C_VEL
LIN {X 0,Y 318.951,Z 344.472,A -85,B 0,C 180,E1 -15333.805,E2 -15333.805} C_VEL
LIN {X 0,Y 319.493,Z 338.518,A -85,B 0,C 180,E1 -15335.52,E2 -15335.52} C_VEL
LIN {X 0,Y 320.165,Z 331.716,A -85,B 0,C 180,E1 -15337.132,E2 -15337.132} C_VEL
LIN {X 0,Y 321.06,Z 321.974,A -85,B 0,C 180,E1 -15339.001,E2 -15339.001} C_VEL
LIN {X 0,Y 322.076,Z 311.357,A -85,B 0,C 180,E1 -15340.635,E2 -15340.635} C_VEL
LIN {X 0,Y 323.017,Z 300.259,A -85,B 0,C 180,E1 -15341.992,E2 -15341.992} C_VEL
LIN {X 0,Y 323.938,Z 287.616,A -85,B 0,C 180,E1 -15343.216,E2 -15343.216} C_VEL
LIN {X 0,Y 324.779,Z 275.286,A -85,B 0,C 180,E1 -15344.113,E2 -15344.113} C_VEL
LIN {X 0,Y 325.281,Z 262.372,A -85,B 0,C 180,E1 -15344.805,E2 -15344.805} C_VEL
LIN {X 0,Y 325.756,Z 248.347,A -85,B 0,C 180,E1 -15345.282,E2 -15345.282} C_VEL
LIN {X 0,Y 327.858,Z 174.518,A -85,B 0,C 180,E1 -15347.237,E2 -15347.237} C_VEL
LIN {X 0,Y 320.279,Z 150.892,A -85,B 0,C 180,E1 -15348.329,E2 -15348.329} C_VEL
LIN {X 0,Y 319.595,Z 148.675,A -85,B 0,C 180,E1 -15348.447,E2 -15348.447} C_VEL
LIN {X 0,Y 319.561,Z 148.677,A -85,B 0,C 180,E1 -15352.347,E2 -15352.347} C_VEL
LIN {X 0,Y 319.559,Z 148.678,A -85,B 0,C 180,E1 -15355.123,E2 -15355.123} C_VEL
LIN {X 0,Y 319.569,Z 148.677,A -85,B 0,C 180,E1 -15359.057,E2 -15359.057} C_VEL
LIN {X 0,Y 319.608,Z 148.67,A -85,B 0,C 180,E1 -15362.498,E2 -15362.498} C_VEL
LIN {X 0,Y 319.605,Z 148.676,A -85,B 0,C 180,E1 -15365.304,E2 -15365.304} C_VEL
LIN {X 0,Y 319.595,Z 148.672,A -85,B 0,C 180,E1 -15368.047,E2 -15368.047} C_VEL
LIN {X 0,Y 319.623,Z 148.668,A -85,B 0,C 180,E1 -15372.071,E2 -15372.071} C_VEL
LIN {X 0,Y 319.731,Z 148.655,A -85,B 0,C 180,E1 -15376.007,E2 -15376.007} C_VEL
LIN {X 0,Y 319.756,Z 148.652,A -85,B 0,C 180,E1 -15379.872,E2 -15379.872} C_VEL
LIN {X 0,Y 319.924,Z 148.632,A -85,B 0,C 180,E1 -15382.426,E2 -15382.426} C_VEL
LIN {X 0,Y 319.744,Z 148.659,A -85,B 0,C 180,E1 -15384.956,E2 -15384.956} C_VEL
LIN {X 0,Y 319.99,Z 148.623,A -85,B 0,C 180,E1 -15387.482,E2 -15387.482} C_VEL
LIN {X 0,Y 320.149,Z 148.603,A -85,B 0,C 180,E1 -15390,E2 -15390} C_VEL
LIN {X 0,Y 319.989,Z 148.626,A -85,B 0,C 180,E1 -15392.517,E2 -15392.517} C_VEL
LIN {X 0,Y 319.943,Z 148.631,A -85,B 0,C 180,E1 -15396.305,E2 -15396.305} C_VEL
LIN {X 0,Y 319.84,Z 148.645,A -85,B 0,C 180,E1 -15398.848,E2 -15398.848} C_VEL
LIN {X 0,Y 319.68,Z 148.665,A -85,B 0,C 180,E1 -15402.699,E2 -15402.699} C_VEL
LIN {X 0,Y 319.697,Z 148.659,A -85,B 0,C 180,E1 -15405.295,E2 -15405.295} C_VEL
LIN {X 0,Y 319.671,Z 148.662,A -85,B 0,C 180,E1 -15409.255,E2 -15409.255} C_VEL
LIN {X 0,Y 319.557,Z 148.676,A -85,B 0,C 180,E1 -15413.32,E2 -15413.32} C_VEL
LIN {X 0,Y 319.632,Z 148.671,A -85,B 0,C 180,E1 -15416.088,E2 -15416.088} C_VEL
LIN {X 0,Y 319.595,Z 148.672,A -85,B 0,C 180,E1 -15418.932,E2 -15418.932} C_VEL
LIN {X 0,Y 319.535,Z 148.682,A -85,B 0,C 180,E1 -15421.861,E2 -15421.861} C_VEL
LIN {X 0,Y 319.577,Z 148.675,A -85,B 0,C 180,E1 -15425.543,E2 -15425.543} C_VEL
LIN {X 0,Y 319.594,Z 148.678,A -85,B 0,C 180,E1 -15428.004,E2 -15428.004} C_VEL
LIN {X 0,Y 319.593,Z 148.675,A -85,B 0,C 180,E1 -15431.611,E2 -15431.611} C_VEL
LIN {X 0,Y 319.598,Z 148.673,A -85,B 0,C 180,E1 -15433.385,E2 -15433.385} C_VEL
LIN {X 0,Y 318.934,Z 148.76,A -85,B 0,C 180,E1 -15434.436,E2 -15434.436} C_VEL
LIN {X 0,Y 316.051,Z 149.118,A -85,B 0,C 180,E1 -15436.144,E2 -15436.144} C_VEL
LIN {X 0,Y 313.606,Z 149.421,A -85,B 0,C 180,E1 -15437.53,E2 -15437.53} C_VEL
LIN {X 0,Y 312.568,Z 149.548,A -85,B 0,C 180,E1 -15438.603,E2 -15438.603} C_VEL
LIN {X 0,Y 312.489,Z 149.557,A -85,B 0,C 180,E1 -15438.967,E2 -15438.967} C_VEL
LIN {X 0,Y 312.537,Z 149.551,A -85,B 0,C 180,E1 -15442.617,E2 -15442.617} C_VEL
LIN {X 0,Y 312.516,Z 149.554,A -85,B 0,C 180,E1 -15446.311,E2 -15446.311} C_VEL
LIN {X 0,Y 312.542,Z 149.55,A -85,B 0,C 180,E1 -15450.35,E2 -15450.35} C_VEL
LIN {X 0,Y 312.599,Z 149.544,A -85,B 0,C 180,E1 -15454.065,E2 -15454.065} C_VEL
LIN {X 0,Y 312.584,Z 149.549,A -85,B 0,C 180,E1 -15457.529,E2 -15457.529} C_VEL
LIN {X 0,Y 312.635,Z 149.541,A -85,B 0,C 180,E1 -15461.657,E2 -15461.657} C_VEL
LIN {X 0,Y 312.691,Z 149.533,A -85,B 0,C 180,E1 -15465.687,E2 -15465.687} C_VEL
LIN {X 0,Y 312.699,Z 149.532,A -85,B 0,C 180,E1 -15469.642,E2 -15469.642} C_VEL
LIN {X 0,Y 312.863,Z 149.511,A -85,B 0,C 180,E1 -15472.255,E2 -15472.255} C_VEL
LIN {X 0,Y 312.714,Z 149.533,A -85,B 0,C 180,E1 -15474.843,E2 -15474.843} C_VEL
LIN {X 0,Y 312.989,Z 149.498,A -85,B 0,C 180,E1 -15478.714,E2 -15478.714} C_VEL
LIN {X 0,Y 312.989,Z 149.496,A -85,B 0,C 180,E1 -15481.287,E2 -15481.287} C_VEL
LIN {X 0,Y 312.717,Z 149.531,A -85,B 0,C 180,E1 -15485.158,E2 -15485.158} C_VEL
LIN {X 0,Y 312.87,Z 149.51,A -85,B 0,C 180,E1 -15487.746,E2 -15487.746} C_VEL
LIN {X 0,Y 312.668,Z 149.534,A -85,B 0,C 180,E1 -15491.672,E2 -15491.672} C_VEL
LIN {X 0,Y 312.698,Z 149.533,A -85,B 0,C 180,E1 -15494.888,E2 -15494.888} C_VEL
LIN {X 0,Y 312.628,Z 149.54,A -85,B 0,C 180,E1 -15499.237,E2 -15499.237} C_VEL
LIN {X 0,Y 312.525,Z 149.555,A -85,B 0,C 180,E1 -15502.781,E2 -15502.781} C_VEL
LIN {X 0,Y 312.601,Z 149.545,A -85,B 0,C 180,E1 -15505.936,E2 -15505.936} C_VEL
LIN {X 0,Y 312.544,Z 149.551,A -85,B 0,C 180,E1 -15509.651,E2 -15509.651} C_VEL
LIN {X 0,Y 312.519,Z 149.555,A -85,B 0,C 180,E1 -15513.69,E2 -15513.69} C_VEL
LIN {X 0,Y 312.551,Z 149.549,A -85,B 0,C 180,E1 -15517.382,E2 -15517.382} C_VEL
LIN {X 0,Y 312.5,Z 149.556,A -85,B 0,C 180,E1 -15520.708,E2 -15520.708} C_VEL
LIN {X 0,Y 312.465,Z 149.563,A -85,B 0,C 180,E1 -15524.208,E2 -15524.208} C_VEL
LIN {X 0,Y 312.484,Z 149.563,A -85,B 0,C 180,E1 -15527.919,E2 -15527.919} C_VEL
LIN {X 0,Y 312.535,Z 149.556,A -85,B 0,C 180,E1 -15531.911,E2 -15531.911} C_VEL
LIN {X 0,Y 312.507,Z 149.56,A -85,B 0,C 180,E1 -15535.791,E2 -15535.791} C_VEL
LIN {X 0,Y 312.563,Z 149.664,A -85,B 0,C 180,E1 -15537.749,E2 -15537.749} C_VEL
LIN {X 0,Y 315.643,Z 164.333,A -85,B 0,C 180,E1 -15541.762,E2 -15541.762} C_VEL
LIN {X 0,Y 316.593,Z 169.741,A -85,B 0,C 180,E1 -15543.191,E2 -15543.191} C_VEL
LIN {X 0,Y 315.578,Z 179.736,A -85,B 0,C 180,E1 -15545.646,E2 -15545.646} C_VEL
LIN {X 0,Y 315.234,Z 182.39,A -85,B 0,C 180,E1 -15546.288,E2 -15546.288} C_VEL
LIN {X 0,Y 320.169,Z 225.06,A -85,B 0,C 180,E1 -15547.802,E2 -15547.802} C_VEL
LIN {X 0,Y 318.352,Z 291.584,A -85,B 0,C 180,E1 -15549.654,E2 -15549.654} C_VEL
LIN {X 0,Y 317.574,Z 305.184,A -85,B 0,C 180,E1 -15550.277,E2 -15550.277} C_VEL
LIN {X 0,Y 316.681,Z 317.181,A -85,B 0,C 180,E1 -15551.061,E2 -15551.061} C_VEL
LIN {X 0,Y 315.681,Z 328.169,A -85,B 0,C 180,E1 -15552.008,E2 -15552.008} C_VEL
LIN {X 0,Y 314.575,Z 339.768,A -85,B 0,C 180,E1 -15553.284,E2 -15553.284} C_VEL
LIN {X 0,Y 313.412,Z 350.72,A -85,B 0,C 180,E1 -15554.793,E2 -15554.793} C_VEL
LIN {X 0,Y 312.632,Z 359.761,A -85,B 0,C 180,E1 -15556.348,E2 -15556.348} C_VEL
LIN {X 0,Y 311.966,Z 367.554,A -85,B 0,C 180,E1 -15557.973,E2 -15557.973} C_VEL
LIN {X 0,Y 311.348,Z 375.166,A -85,B 0,C 180,E1 -15559.925,E2 -15559.925} C_VEL
LIN {X 0,Y 311.095,Z 380.314,A -85,B 0,C 180,E1 -15561.556,E2 -15561.556} C_VEL
LIN {X 0,Y 310.915,Z 385.258,A -85,B 0,C 180,E1 -15563.511,E2 -15563.511} C_VEL
LIN {X 0,Y 310.914,Z 388.99,A -85,B 0,C 180,E1 -15565.463,E2 -15565.463} C_VEL
LIN {X 0,Y 310.89,Z 391.609,A -85,B 0,C 180,E1 -15567.409,E2 -15567.409} C_VEL
LIN {X 0,Y 311.006,Z 392.813,A -85,B 0,C 180,E1 -15568.706,E2 -15568.706} C_VEL
LIN {X 0,Y 311.076,Z 393.537,A -85,B 0,C 180,E1 -15570,E2 -15570} C_VEL
LIN {X 0,Y 310.879,Z 393.808,A -85,B 0,C 180,E1 -15571.296,E2 -15571.296} C_VEL
LIN {X 0,Y 310.786,Z 393.674,A -85,B 0,C 180,E1 -15572.593,E2 -15572.593} C_VEL
LIN {X 0,Y 310.767,Z 393.128,A -85,B 0,C 180,E1 -15573.891,E2 -15573.891} C_VEL
LIN {X 0,Y 310.725,Z 391.702,A -85,B 0,C 180,E1 -15575.615,E2 -15575.615} C_VEL
LIN {X 0,Y 310.961,Z 388.85,A -85,B 0,C 180,E1 -15577.794,E2 -15577.794} C_VEL
LIN {X 0,Y 311.366,Z 385.198,A -85,B 0,C 180,E1 -15579.747,E2 -15579.747} C_VEL
LIN {X 0,Y 312.041,Z 380.471,A -85,B 0,C 180,E1 -15581.696,E2 -15581.696} C_VEL
LIN {X 0,Y 313.406,Z 373.386,A -85,B 0,C 180,E1 -15583.95,E2 -15583.95} C_VEL
LIN {X 0,Y 314.722,Z 365.703,A -85,B 0,C 180,E1 -15585.886,E2 -15585.886} C_VEL
LIN {X 0,Y 316.589,Z 356.319,A -85,B 0,C 180,E1 -15587.773,E2 -15587.773} C_VEL
LIN {X 0,Y 318.677,Z 345.535,A -85,B 0,C 180,E1 -15589.486,E2 -15589.486} C_VEL
LIN {X 0,Y 320.703,Z 334.756,A -85,B 0,C 180,E1 -15590.862,E2 -15590.862} C_VEL
LIN {X 0,Y 322.614,Z 322.759,A -85,B 0,C 180,E1 -15592.073,E2 -15592.073} C_VEL
LIN {X 0,Y 324.388,Z 310.286,A -85,B 0,C 180,E1 -15593.038,E2 -15593.038} C_VEL
LIN {X 0,Y 325.985,Z 296.597,A -85,B 0,C 180,E1 -15593.802,E2 -15593.802} C_VEL
LIN {X 0,Y 327.022,Z 282.572,A -85,B 0,C 180,E1 -15594.33,E2 -15594.33} C_VEL
LIN {X 0,Y 329.647,Z 226.371,A -85,B 0,C 180,E1 -15595.97,E2 -15595.97} C_VEL
LIN {X 0,Y 327.506,Z 208.909,A -85,B 0,C 180,E1 -15596.88,E2 -15596.88} C_VEL
LIN {X 0,Y 324.228,Z 191.347,A -85,B 0,C 180,E1 -15597.978,E2 -15597.978} C_VEL
LIN {X 0,Y 321.841,Z 181.55,A -85,B 0,C 180,E1 -15598.713,E2 -15598.713} C_VEL
LIN {X 0,Y 319.675,Z 176.864,A -85,B 0,C 180,E1 -15599.234,E2 -15599.234} C_VEL
LIN {X 0,Y 317.852,Z 168.127,A -85,B 0,C 180,E1 -15602.051,E2 -15602.051} C_VEL
LIN {X 0,Y 315.668,Z 159.889,A -85,B 0,C 180,E1 -15605.007,E2 -15605.007} C_VEL
LIN {X 0,Y 313.676,Z 153.331,A -85,B 0,C 180,E1 -15607.628,E2 -15607.628} C_VEL
LIN {X 0,Y 312.528,Z 149.559,A -85,B 0,C 180,E1 -15609.324,E2 -15609.324} C_VEL
LIN {X 0,Y 312.494,Z 149.558,A -85,B 0,C 180,E1 -15612.432,E2 -15612.432} C_VEL
LIN {X 0,Y 312.462,Z 149.559,A -85,B 0,C 180,E1 -15616.035,E2 -15616.035} C_VEL
LIN {X 0,Y 312.507,Z 149.555,A -85,B 0,C 180,E1 -15619.875,E2 -15619.875} C_VEL
LIN {X 0,Y 312.54,Z 149.548,A -85,B 0,C 180,E1 -15622.616,E2 -15622.616} C_VEL
LIN {X 0,Y 312.523,Z 149.547,A -85,B 0,C 180,E1 -15626.311,E2 -15626.311} C_VEL
LIN {X 0,Y 312.542,Z 149.553,A -85,B 0,C 180,E1 -15630.349,E2 -15630.349} C_VEL
LIN {X 0,Y 312.6,Z 149.539,A -85,B 0,C 180,E1 -15634.066,E2 -15634.066} C_VEL
LIN {X 0,Y 312.591,Z 149.543,A -85,B 0,C 180,E1 -15637.529,E2 -15637.529} C_VEL
LIN {X 0,Y 312.592,Z 149.542,A -85,B 0,C 180,E1 -15641.653,E2 -15641.653} C_VEL
LIN {X 0,Y 312.689,Z 149.536,A -85,B 0,C 180,E1 -15645.685,E2 -15645.685} C_VEL
LIN {X 0,Y 312.689,Z 149.538,A -85,B 0,C 180,E1 -15649.641,E2 -15649.641} C_VEL
LIN {X 0,Y 312.842,Z 149.564,A -85,B 0,C 180,E1 -15652.902,E2 -15652.902} C_VEL
LIN {X 0,Y 314.145,Z 154.253,A -85,B 0,C 180,E1 -15654.926,E2 -15654.926} C_VEL
LIN {X 0,Y 316.736,Z 158.281,A -85,B 0,C 180,E1 -15655.545,E2 -15655.545} C_VEL
LIN {X 0,Y 321.85,Z 166.399,A -85,B 0,C 180,E1 -15656.695,E2 -15656.695} C_VEL
LIN {X 0,Y 326.701,Z 175.552,A -85,B 0,C 180,E1 -15657.778,E2 -15657.778} C_VEL
LIN {X 0,Y 331.303,Z 186.028,A -85,B 0,C 180,E1 -15658.784,E2 -15658.784} C_VEL
LIN {X 0,Y 331.308,Z 190.013,A -85,B 0,C 180,E1 -15658.93,E2 -15658.93} C_VEL
LIN {X 0,Y 327.495,Z 261.146,A -85,B 0,C 180,E1 -15661.037,E2 -15661.037} C_VEL
LIN {X 0,Y 326.56,Z 274.551,A -85,B 0,C 180,E1 -15661.695,E2 -15661.695} C_VEL
LIN {X 0,Y 325.268,Z 287.243,A -85,B 0,C 180,E1 -15662.576,E2 -15662.576} C_VEL
LIN {X 0,Y 323.617,Z 299.831,A -85,B 0,C 180,E1 -15663.735,E2 -15663.735} C_VEL
LIN {X 0,Y 321.913,Z 310.622,A -85,B 0,C 180,E1 -15665.009,E2 -15665.009} C_VEL
LIN {X 0,Y 320.027,Z 321.145,A -85,B 0,C 180,E1 -15666.573,E2 -15666.573} C_VEL
LIN {X 0,Y 318.216,Z 330.264,A -85,B 0,C 180,E1 -15668.253,E2 -15668.253} C_VEL
LIN {X 0,Y 316.431,Z 338.791,A -85,B 0,C 180,E1 -15670.234,E2 -15670.234} C_VEL
LIN {X 0,Y 314.863,Z 345.639,A -85,B 0,C 180,E1 -15672.242,E2 -15672.242} C_VEL
LIN {X 0,Y 313.635,Z 351.001,A -85,B 0,C 180,E1 -15674.269,E2 -15674.269} C_VEL
LIN {X 0,Y 312.641,Z 355.073,A -85,B 0,C 180,E1 -15676.319,E2 -15676.319} C_VEL
LIN {X 0,Y 311.724,Z 358.372,A -85,B 0,C 180,E1 -15678.752,E2 -15678.752} C_VEL
LIN {X 0,Y 311.17,Z 360.177,A -85,B 0,C 180,E1 -15681.184,E2 -15681.184} C_VEL
LIN {X 0,Y 310.948,Z 360.51,A -85,B 0,C 180,E1 -15682.596,E2 -15682.596} C_VEL
LIN {X 0,Y 310.799,Z 360.375,A -85,B 0,C 180,E1 -15684.018,E2 -15684.018} C_VEL
LIN {X 0,Y 310.727,Z 359.723,A -85,B 0,C 180,E1 -15685.451,E2 -15685.451} C_VEL
LIN {X 0,Y 310.716,Z 358.534,A -85,B 0,C 180,E1 -15686.896,E2 -15686.896} C_VEL
LIN {X 0,Y 310.978,Z 355.747,A -85,B 0,C 180,E1 -15689.07,E2 -15689.07} C_VEL
LIN {X 0,Y 311.319,Z 351.584,A -85,B 0,C 180,E1 -15691.28,E2 -15691.28} C_VEL
LIN {X 0,Y 311.769,Z 345.921,A -85,B 0,C 180,E1 -15693.481,E2 -15693.481} C_VEL
LIN {X 0,Y 312.396,Z 339.604,A -85,B 0,C 180,E1 -15695.401,E2 -15695.401} C_VEL
LIN {X 0,Y 313.126,Z 331.842,A -85,B 0,C 180,E1 -15697.301,E2 -15697.301} C_VEL
LIN {X 0,Y 314.055,Z 322.031,A -85,B 0,C 180,E1 -15699.211,E2 -15699.211} C_VEL
LIN {X 0,Y 315.092,Z 311.587,A -85,B 0,C 180,E1 -15700.846,E2 -15700.846} C_VEL
LIN {X 0,Y 316.062,Z 300.431,A -85,B 0,C 180,E1 -15702.236,E2 -15702.236} C_VEL
LIN {X 0,Y 316.963,Z 288.483,A -85,B 0,C 180,E1 -15703.421,E2 -15703.421} C_VEL
LIN {X 0,Y 317.851,Z 275.913,A -85,B 0,C 180,E1 -15704.367,E2 -15704.367} C_VEL
LIN {X 0,Y 318.398,Z 262.349,A -85,B 0,C 180,E1 -15705.11,E2 -15705.11} C_VEL
LIN {X 0,Y 318.864,Z 248.722,A -85,B 0,C 180,E1 -15705.581,E2 -15705.581} C_VEL
LIN {X 0,Y 320.998,Z 175.557,A -85,B 0,C 180,E1 -15707.569,E2 -15707.569} C_VEL
LIN {X 0,Y 313.898,Z 153.674,A -85,B 0,C 180,E1 -15708.609,E2 -15708.609} C_VEL
LIN {X 0,Y 312.519,Z 149.555,A -85,B 0,C 180,E1 -15708.815,E2 -15708.815} C_VEL
LIN {X 0,Y 312.525,Z 149.553,A -85,B 0,C 180,E1 -15712.614,E2 -15712.614} C_VEL
LIN {X 0,Y 312.519,Z 149.554,A -85,B 0,C 180,E1 -15716.311,E2 -15716.311} C_VEL
LIN {X 0,Y 312.545,Z 149.55,A -85,B 0,C 180,E1 -15720.35,E2 -15720.35} C_VEL
LIN {X 0,Y 312.602,Z 149.544,A -85,B 0,C 180,E1 -15724.064,E2 -15724.064} C_VEL
